C09143=1199.165,141.254,-53.045,-178.295,6.103,148.591
C09144=1199.160,141.502,-53.066,-178.292,6.105,148.590
C09145=1199.155,141.752,-53.087,-178.290,6.105,148.590
C09146=1199.151,142.001,-53.107,-178.287,6.107,148.589
C09147=1199.145,142.250,-53.128,-178.285,6.109,148.589
C09148=1199.141,142.499,-53.148,-178.282,6.110,148.589
C09149=1199.136,142.748,-53.169,-178.279,6.111,148.588
C09150=1199.131,142.997,-53.190,-178.277,6.113,148.588
C09151=1199.127,143.246,-53.210,-178.274,6.114,148.587
C09152=1199.122,143.495,-53.231,-178.272,6.116,148.587
C09153=1199.117,143.744,-53.251,-178.269,6.117,148.586
C09154=1199.112,143.994,-53.272,-178.266,6.118,148.586
C09155=1199.108,144.243,-53.293,-178.264,6.120,148.586
C09156=1199.103,144.492,-53.314,-178.261,6.122,148.585
C09157=1199.099,144.741,-53.335,-178.259,6.122,148.585
C09158=1199.094,144.990,-53.356,-178.256,6.124,148.584
C09159=1199.089,145.239,-53.376,-178.253,6.126,148.584
C09160=1199.084,145.488,-53.397,-178.251,6.126,148.583
C09161=1199.080,145.737,-53.418,-178.248,6.128,148.583
C09162=1199.075,145.986,-53.439,-178.245,6.130,148.582
C09163=1199.070,146.235,-53.459,-178.243,6.132,148.582
C09164=1199.065,146.484,-53.481,-178.240,6.132,148.581
C09165=1199.060,146.733,-53.502,-178.237,6.134,148.581
C09166=1199.056,146.983,-53.522,-178.235,6.136,148.581
C09167=1199.051,147.232,-53.543,-178.232,6.137,148.580
C09168=1199.047,147.481,-53.564,-178.230,6.139,148.580
C09169=1199.042,147.730,-53.585,-178.227,6.140,148.579
C09170=1199.037,147.979,-53.606,-178.224,6.141,148.579
C09171=1199.032,148.228,-53.627,-178.222,6.143,148.578
C09172=1199.027,148.477,-53.648,-178.219,6.145,148.578
C09173=1199.023,148.726,-53.669,-178.217,6.145,148.577
C09174=1199.018,148.976,-53.690,-178.214,6.147,148.577
C09175=1199.013,149.225,-53.711,-178.211,6.149,148.577
C09176=1199.009,149.473,-53.732,-178.208,6.151,148.576
C09177=1199.004,149.722,-53.753,-178.206,6.151,148.576
C09178=1198.999,149.972,-53.774,-178.203,6.153,148.575
C09179=1198.994,150.220,-53.795,-178.201,6.155,148.575
C09180=1198.990,150.470,-53.817,-178.198,6.156,148.575
C09181=1198.985,150.719,-53.838,-178.195,6.157,148.574
C09182=1198.981,150.968,-53.859,-178.193,6.159,148.574
C09183=1198.975,151.217,-53.880,-178.190,6.161,148.573
C09184=1198.970,151.466,-53.901,-178.188,6.162,148.573
C09185=1198.967,151.715,-53.922,-178.185,6.163,148.572
C09186=1198.961,151.964,-53.943,-178.182,6.165,148.572
C09187=1198.957,152.213,-53.965,-178.180,6.166,148.571
C09188=1198.952,152.462,-53.985,-178.177,6.168,148.571
C09189=1198.947,152.711,-54.006,-178.174,6.169,148.571
C09190=1198.943,152.961,-54.028,-178.172,6.171,148.570
C09191=1198.938,153.210,-54.049,-178.169,6.172,148.570
C09192=1198.933,153.458,-54.070,-178.167,6.174,148.569
C09193=1198.928,153.707,-54.091,-178.164,6.175,148.569
C09194=1198.924,153.957,-54.113,-178.161,6.177,148.569
C09195=1198.919,154.206,-54.134,-178.159,6.178,148.568
C09196=1198.914,154.455,-54.156,-178.156,6.180,148.568
C09197=1198.910,154.704,-54.176,-178.153,6.181,148.567
C09198=1198.905,154.953,-54.198,-178.151,6.183,148.567
C09199=1198.900,155.202,-54.219,-178.148,6.184,148.566
C09200=1198.895,155.451,-54.241,-178.146,6.186,148.566
C09201=1198.890,155.699,-54.263,-178.143,6.187,148.565
C09202=1198.887,155.949,-54.283,-178.140,6.189,148.565
C09203=1198.882,156.198,-54.305,-178.138,6.190,148.565
C09204=1198.876,156.447,-54.326,-178.135,6.192,148.564
C09205=1198.872,156.696,-54.348,-178.132,6.194,148.564
C09206=1198.867,156.945,-54.370,-178.129,6.195,148.563
C09207=1198.862,157.194,-54.391,-178.127,6.196,148.563
C09208=1198.858,157.443,-54.412,-178.125,6.198,148.563
C09209=1198.853,157.693,-54.433,-178.122,6.200,148.562
C09210=1198.849,157.941,-54.455,-178.119,6.201,148.562
C09211=1198.844,158.190,-54.476,-178.117,6.202,148.561
C09212=1198.839,158.440,-54.498,-178.114,6.204,148.561
C09213=1198.835,158.708,-54.521,-178.111,6.206,148.560
C09214=1198.829,158.978,-54.545,-178.109,6.207,148.560
C09215=1198.823,159.246,-54.568,-178.105,6.209,148.559
C09216=1198.819,159.515,-54.591,-178.103,6.211,148.559
C09217=1198.814,159.765,-54.612,-178.100,6.212,148.559
C09218=1198.809,160.013,-54.634,-178.097,6.214,148.558
C09219=1198.804,160.262,-54.656,-178.095,6.215,148.558
C09220=1198.800,160.511,-54.678,-178.092,6.217,148.557
C09221=1198.795,160.760,-54.699,-178.089,6.218,148.557
C09222=1198.791,161.010,-54.721,-178.087,6.220,148.557
C09223=1198.786,161.258,-54.743,-178.084,6.222,148.556
C09224=1198.781,161.507,-54.764,-178.082,6.223,148.556
C09225=1198.777,161.756,-54.786,-178.079,6.225,148.556
C09226=1198.771,162.006,-54.807,-178.076,6.226,148.555
C09227=1198.767,162.254,-54.829,-178.073,6.228,148.555
C09228=1198.762,162.504,-54.851,-178.071,6.230,148.554
C09229=1198.757,162.752,-54.873,-178.069,6.231,148.554
C09230=1198.753,163.002,-54.895,-178.066,6.233,148.553
C09231=1198.748,163.250,-54.916,-178.063,6.234,148.553
C09232=1198.744,163.500,-54.938,-178.061,6.236,148.553
C09233=1198.739,163.748,-54.960,-178.058,6.238,148.552
C09234=1198.734,163.998,-54.981,-178.055,6.239,148.552
C09235=1198.730,164.247,-55.003,-178.053,6.240,148.551
C09236=1198.725,164.496,-55.025,-178.050,6.242,148.551
C09237=1198.721,164.745,-55.047,-178.047,6.244,148.551
C09238=1198.716,164.994,-55.069,-178.045,6.246,148.550
C09239=1198.711,165.243,-55.091,-178.043,6.247,148.550
C09240=1198.707,165.492,-55.112,-178.039,6.248,148.549
C09241=1198.702,165.740,-55.134,-178.037,6.250,148.549
C09242=1198.697,165.989,-55.156,-178.034,6.252,148.549
C09243=1198.692,166.238,-55.178,-178.031,6.254,148.548
C09244=1198.688,166.488,-55.200,-178.029,6.255,148.548
C09245=1198.683,166.736,-55.222,-178.027,6.256,148.547
C09246=1198.678,166.986,-55.244,-178.024,6.258,148.547
C09247=1198.674,167.234,-55.266,-178.021,6.260,148.547
C09248=1198.669,167.484,-55.288,-178.019,6.262,148.546
C09249=1198.664,167.732,-55.309,-178.016,6.263,148.546
C09250=1198.660,167.981,-55.333,-178.013,6.264,148.545
C09251=1198.655,168.230,-55.355,-178.011,6.266,148.545
C09252=1198.651,168.479,-55.377,-178.008,6.268,148.545
C09253=1198.646,168.728,-55.398,-178.005,6.270,148.544
C09254=1198.641,168.977,-55.420,-178.003,6.271,148.544
C09255=1198.636,169.226,-55.443,-178.000,6.273,148.544
C09256=1198.632,169.476,-55.465,-177.998,6.274,148.543
C09257=1198.627,169.724,-55.486,-177.995,6.276,148.543
C09258=1198.623,169.973,-55.509,-177.992,6.277,148.542
C09259=1198.618,170.222,-55.531,-177.989,6.279,148.542
C09260=1198.613,170.471,-55.553,-177.987,6.281,148.541
C09261=1198.608,170.720,-55.575,-177.984,6.283,148.541
C09262=1198.604,170.969,-55.597,-177.981,6.285,148.541
C09263=1198.599,171.217,-55.620,-177.979,6.285,148.540
C09264=1198.594,171.467,-55.642,-177.977,6.287,148.540
C09265=1198.590,171.716,-55.664,-177.974,6.289,148.540
C09266=1198.585,171.965,-55.686,-177.971,6.291,148.539
C09267=1198.580,172.214,-55.709,-177.969,6.293,148.539
C09268=1198.575,172.463,-55.731,-177.966,6.294,148.539
C09269=1198.571,172.712,-55.753,-177.963,6.296,148.538
C09270=1198.566,172.961,-55.775,-177.961,6.297,148.538
C09271=1198.562,173.210,-55.798,-177.958,6.299,148.537
C09272=1198.557,173.459,-55.820,-177.955,6.300,148.537
C09273=1198.553,173.708,-55.842,-177.953,6.302,148.536
C09274=1198.548,173.957,-55.865,-177.950,6.304,148.536
C09275=1198.543,174.205,-55.887,-177.947,6.306,148.536
C09276=1198.539,174.455,-55.909,-177.945,6.308,148.535
C09277=1198.534,174.704,-55.932,-177.943,6.309,148.535
C09278=1198.529,174.952,-55.954,-177.940,6.310,148.535
C09279=1198.524,175.201,-55.977,-177.937,6.312,148.534
C09280=1198.520,175.451,-55.999,-177.935,6.314,148.534
C09281=1198.515,175.699,-56.021,-177.932,6.316,148.534
C09282=1198.511,175.948,-56.044,-177.929,6.318,148.533
C09283=1198.506,176.197,-56.066,-177.927,6.319,148.533
C09284=1198.501,176.446,-56.089,-177.924,6.321,148.532
C09285=1198.497,176.695,-56.111,-177.921,6.323,148.532
C09286=1198.492,176.943,-56.134,-177.919,6.324,148.531
C09287=1198.487,177.193,-56.156,-177.916,6.325,148.531
C09288=1198.483,177.442,-56.179,-177.913,6.327,148.531
C09289=1198.478,177.691,-56.201,-177.911,6.329,148.530
C09290=1198.474,177.939,-56.224,-177.908,6.331,148.530
C09291=1198.469,178.189,-56.247,-177.905,6.333,148.530
C09292=1198.464,178.437,-56.269,-177.903,6.334,148.529
C09293=1198.459,178.687,-56.292,-177.900,6.336,148.529
C09294=1198.455,178.935,-56.315,-177.897,6.338,148.529
C09295=1198.450,179.185,-56.337,-177.895,6.340,148.528
C09296=1198.446,179.433,-56.360,-177.893,6.341,148.528
C09297=1198.441,179.682,-56.382,-177.890,6.343,148.528
C09298=1198.437,179.932,-56.405,-177.887,6.344,148.527
C09299=1198.431,180.180,-56.428,-177.885,6.346,148.527
C09300=1198.427,180.429,-56.450,-177.882,6.348,148.526
C09301=1198.422,180.678,-56.474,-177.879,6.350,148.526
C09302=1198.418,180.927,-56.496,-177.877,6.352,148.526
C09303=1198.413,181.176,-56.519,-177.874,6.353,148.525
C09304=1198.409,181.425,-56.541,-177.871,6.355,148.525
C09305=1198.404,181.674,-56.565,-177.869,6.357,148.525
C09306=1198.400,181.923,-56.587,-177.866,6.359,148.524
C09307=1198.394,182.171,-56.610,-177.863,6.361,148.524
C09308=1198.391,182.420,-56.633,-177.861,6.362,148.524
C09309=1198.386,182.670,-56.655,-177.859,6.363,148.523
C09310=1198.381,182.919,-56.679,-177.856,6.365,148.523
C09311=1198.376,183.167,-56.701,-177.853,6.367,148.522
C09312=1198.372,183.416,-56.724,-177.851,6.369,148.522
C09313=1198.367,183.665,-56.746,-177.848,6.371,148.522
C09314=1198.363,183.914,-56.770,-177.845,6.373,148.521
C09315=1198.358,184.163,-56.793,-177.843,6.374,148.521
C09316=1198.353,184.411,-56.815,-177.840,6.376,148.521
C09317=1198.348,184.681,-56.840,-177.837,6.378,148.520
C09318=1198.343,184.951,-56.866,-177.834,6.379,148.520
C09319=1198.338,185.220,-56.890,-177.831,6.381,148.519
C09320=1198.333,185.490,-56.915,-177.828,6.384,148.519
C09321=1198.328,185.739,-56.938,-177.826,6.386,148.519
C09322=1198.324,185.988,-56.961,-177.823,6.387,148.518
C09323=1198.319,186.237,-56.984,-177.820,6.389,148.518
C09324=1198.315,186.486,-57.008,-177.818,6.390,148.518
C09325=1198.310,186.734,-57.030,-177.816,6.392,148.517
C09326=1198.305,186.983,-57.053,-177.813,6.394,148.517
C09327=1198.300,187.232,-57.076,-177.810,6.396,148.517
C09328=1198.296,187.482,-57.100,-177.808,6.397,148.516
C09329=1198.292,187.730,-57.122,-177.805,6.399,148.516
C09330=1198.287,187.979,-57.146,-177.802,6.401,148.516
C09331=1198.282,188.228,-57.169,-177.800,6.403,148.515
C09332=1198.277,188.477,-57.192,-177.797,6.405,148.515
C09333=1198.273,188.725,-57.215,-177.794,6.406,148.514
C09334=1198.268,188.974,-57.238,-177.792,6.408,148.514
C09335=1198.264,189.223,-57.262,-177.789,6.410,148.514
C09336=1198.259,189.472,-57.285,-177.786,6.412,148.513
C09337=1198.255,189.721,-57.308,-177.784,6.414,148.513
C09338=1198.250,189.970,-57.331,-177.781,6.416,148.513
C09339=1198.246,190.219,-57.354,-177.778,6.417,148.512
C09340=1198.241,190.468,-57.378,-177.776,6.419,148.512
C09341=1198.236,190.717,-57.401,-177.773,6.421,148.512
C09342=1198.231,190.966,-57.424,-177.771,6.423,148.512
C09343=1198.227,191.214,-57.447,-177.768,6.425,148.511
C09344=1198.222,191.463,-57.470,-177.765,6.427,148.511
C09345=1198.218,191.712,-57.494,-177.763,6.429,148.511
C09346=1198.213,191.961,-57.518,-177.760,6.430,148.510
C09347=1198.209,192.210,-57.541,-177.757,6.432,148.510
C09348=1198.204,192.459,-57.564,-177.755,6.434,148.509
C09349=1198.199,192.708,-57.588,-177.752,6.436,148.509
C09350=1198.194,192.957,-57.611,-177.750,6.438,148.509
C09351=1198.190,193.206,-57.634,-177.747,6.439,148.508
C09352=1198.186,193.454,-57.658,-177.744,6.441,148.508
C09353=1198.181,193.703,-57.681,-177.742,6.443,148.508
C09354=1198.177,193.952,-57.705,-177.739,6.445,148.507
C09355=1198.172,194.201,-57.728,-177.736,6.447,148.507
C09356=1198.168,194.450,-57.752,-177.734,6.448,148.507
C09357=1198.163,194.699,-57.775,-177.731,6.450,148.506
C09358=1198.158,194.948,-57.799,-177.728,6.452,148.506
C09359=1198.153,195.197,-57.822,-177.726,6.454,148.506
C09360=1198.149,195.445,-57.846,-177.723,6.456,148.505
C09361=1198.144,195.694,-57.870,-177.721,6.458,148.505
C09362=1198.140,195.943,-57.893,-177.718,6.460,148.505
C09363=1198.135,196.192,-57.917,-177.715,6.461,148.504
C09364=1198.131,196.441,-57.940,-177.713,6.463,148.504
C09365=1198.126,196.690,-57.964,-177.710,6.465,148.504
C09366=1198.121,196.938,-57.988,-177.707,6.467,148.503
C09367=1198.117,197.187,-58.011,-177.705,6.469,148.503
C09368=1198.112,197.436,-58.035,-177.702,6.471,148.503
C09369=1198.108,197.685,-58.059,-177.700,6.472,148.502
C09370=1198.103,197.934,-58.082,-177.697,6.474,148.502
C09371=1198.098,198.183,-58.105,-177.695,6.476,148.502
C09372=1198.094,198.431,-58.129,-177.692,6.478,148.502
C09373=1198.089,198.680,-58.153,-177.689,6.480,148.501
C09374=1198.085,198.928,-58.177,-177.687,6.482,148.501
C09375=1198.080,199.177,-58.200,-177.684,6.484,148.501
C09376=1198.076,199.426,-58.224,-177.681,6.485,148.500
C09377=1198.070,199.675,-58.248,-177.679,6.487,148.500
C09378=1198.066,199.924,-58.272,-177.676,6.490,148.500
C09379=1198.061,200.173,-58.296,-177.673,6.492,148.499
C09380=1198.057,200.421,-58.320,-177.670,6.493,148.499
C09381=1198.053,200.671,-58.343,-177.668,6.496,148.499
C09382=1198.048,200.919,-58.368,-177.665,6.497,148.498
C09383=1198.044,201.168,-58.391,-177.663,6.499,148.498
C09384=1198.039,201.417,-58.415,-177.660,6.501,148.498
C09385=1198.034,201.666,-58.439,-177.657,6.503,148.497
C09386=1198.029,201.914,-58.463,-177.655,6.505,148.497
C09387=1198.025,202.163,-58.486,-177.652,6.506,148.497
C09388=1198.020,202.412,-58.510,-177.649,6.508,148.496
C09389=1198.016,202.661,-58.535,-177.647,6.510,148.496
C09390=1198.012,202.910,-58.558,-177.645,6.512,148.496
C09391=1198.007,203.159,-58.583,-177.642,6.514,148.495
C09392=1198.002,203.408,-58.606,-177.639,6.516,148.495
C09393=1197.998,203.656,-58.630,-177.637,6.518,148.495
C09394=1197.993,203.905,-58.654,-177.634,6.520,148.494
C09395=1197.988,204.154,-58.678,-177.631,6.522,148.494
C09396=1197.984,204.403,-58.703,-177.628,6.524,148.494
C09397=1197.980,204.652,-58.727,-177.626,6.526,148.494
C09398=1197.975,204.900,-58.751,-177.623,6.528,148.493
C09399=1197.970,205.149,-58.775,-177.621,6.530,148.493
C09400=1197.965,205.398,-58.799,-177.618,6.532,148.493
C09401=1197.962,205.647,-58.823,-177.615,6.533,148.492
C09402=1197.957,205.896,-58.847,-177.613,6.535,148.492
C09403=1197.952,206.145,-58.871,-177.610,6.537,148.492
C09404=1197.947,206.393,-58.896,-177.608,6.539,148.492
C09405=1197.943,206.641,-58.920,-177.605,6.541,148.491
C09406=1197.938,206.891,-58.945,-177.602,6.544,148.491
C09407=1197.934,207.140,-58.968,-177.599,6.545,148.491
C09408=1197.929,207.388,-58.992,-177.597,6.547,148.490
C09409=1197.924,207.637,-59.017,-177.594,6.549,148.490
C09410=1197.920,207.885,-59.041,-177.592,6.551,148.490
C09411=1197.916,208.134,-59.065,-177.589,6.553,148.489
C09412=1197.911,208.383,-59.090,-177.587,6.555,148.489
C09413=1197.906,208.632,-59.113,-177.584,6.557,148.489
C09414=1197.902,208.881,-59.137,-177.581,6.559,148.488
C09415=1197.897,209.130,-59.162,-177.579,6.560,148.488
C09416=1197.893,209.378,-59.186,-177.576,6.563,148.488
C09417=1197.888,209.627,-59.211,-177.573,6.565,148.488
C09418=1197.883,209.876,-59.235,-177.571,6.567,148.487
C09419=1197.879,210.125,-59.260,-177.568,6.569,148.487
C09420=1197.874,210.373,-59.284,-177.565,6.571,148.487
C09421=1197.869,210.644,-59.311,-177.563,6.572,148.486
C09422=1197.864,210.914,-59.336,-177.559,6.575,148.486
C09423=1197.860,211.185,-59.363,-177.557,6.577,148.486
C09424=1197.855,211.455,-59.390,-177.554,6.580,148.485
C09425=1197.850,211.704,-59.415,-177.551,6.582,148.485
C09426=1197.845,211.952,-59.439,-177.549,6.584,148.485
C09427=1197.841,212.202,-59.464,-177.546,6.585,148.485
C09428=1197.836,212.450,-59.488,-177.544,6.587,148.484
C09429=1197.831,212.699,-59.513,-177.541,6.589,148.484
C09430=1197.827,212.948,-59.537,-177.539,6.591,148.484
C09431=1197.822,213.197,-59.562,-177.536,6.593,148.483
C09432=1197.818,213.445,-59.586,-177.533,6.596,148.483
C09433=1197.814,213.694,-59.612,-177.530,6.597,148.483
C09434=1197.809,213.942,-59.636,-177.528,6.599,148.482
C09435=1197.804,214.191,-59.660,-177.525,6.601,148.482
C09436=1197.800,214.440,-59.685,-177.523,6.603,148.482
C09437=1197.795,214.689,-59.710,-177.520,6.605,148.482
C09438=1197.791,214.938,-59.734,-177.517,6.607,148.481
C09439=1197.786,215.187,-59.759,-177.514,6.610,148.481
C09440=1197.782,215.434,-59.783,-177.512,6.612,148.481
C09441=1197.778,215.684,-59.808,-177.509,6.614,148.481
C09442=1197.773,215.933,-59.833,-177.507,6.615,148.480
C09443=1197.768,216.181,-59.857,-177.504,6.617,148.480
C09444=1197.764,216.430,-59.882,-177.501,6.619,148.480
C09445=1197.760,216.678,-59.907,-177.499,6.622,148.479
C09446=1197.755,216.928,-59.932,-177.496,6.624,148.479
C09447=1197.750,217.176,-59.957,-177.493,6.626,148.479
C09448=1197.746,217.424,-59.982,-177.491,6.627,148.478
C09449=1197.741,217.674,-60.007,-177.489,6.630,148.478
C09450=1197.736,217.922,-60.031,-177.486,6.631,148.478
C09451=1197.732,218.171,-60.056,-177.483,6.634,148.478
C09452=1197.727,218.420,-60.081,-177.480,6.636,148.477
C09453=1197.723,218.669,-60.106,-177.478,6.638,148.477
C09454=1197.719,218.917,-60.130,-177.475,6.640,148.477
C09455=1197.714,219.166,-60.156,-177.473,6.642,148.477
C09456=1197.709,219.415,-60.181,-177.470,6.644,148.476
C09457=1197.705,219.663,-60.205,-177.467,6.647,148.476
C09458=1197.701,219.912,-60.230,-177.465,6.648,148.476
C09459=1197.695,220.161,-60.255,-177.462,6.650,148.476
C09460=1197.692,220.409,-60.280,-177.459,6.652,148.475
C09461=1197.687,220.658,-60.305,-177.457,6.654,148.475
C09462=1197.683,220.907,-60.331,-177.455,6.656,148.475
C09463=1197.677,221.156,-60.355,-177.451,6.659,148.474
C09464=1197.674,221.404,-60.380,-177.449,6.660,148.474
C09465=1197.669,221.653,-60.405,-177.447,6.663,148.474
C09466=1197.664,221.902,-60.430,-177.444,6.664,148.474
C09467=1197.660,222.150,-60.456,-177.441,6.666,148.473
C09468=1197.655,222.400,-60.481,-177.438,6.669,148.473
C09469=1197.651,222.648,-60.505,-177.436,6.671,148.473
C09470=1197.647,222.896,-60.531,-177.433,6.673,148.473
C09471=1197.642,223.145,-60.556,-177.431,6.675,148.472
C09472=1197.637,223.394,-60.582,-177.428,6.677,148.472
C09473=1197.632,223.643,-60.606,-177.426,6.679,148.472
C09474=1197.629,223.891,-60.631,-177.423,6.681,148.472
C09475=1197.624,224.140,-60.656,-177.420,6.683,148.471
C09476=1197.619,224.389,-60.682,-177.418,6.685,148.471
C09477=1197.615,224.637,-60.707,-177.415,6.687,148.471
C09478=1197.610,224.886,-60.732,-177.412,6.689,148.470
C09479=1197.606,225.135,-60.758,-177.410,6.692,148.470
C09480=1197.601,225.384,-60.783,-177.407,6.694,148.470
C09481=1197.597,225.632,-60.808,-177.404,6.696,148.470
C09482=1197.592,225.880,-60.833,-177.402,6.698,148.470
C09483=1197.588,226.130,-60.858,-177.400,6.700,148.469
C09484=1197.583,226.378,-60.884,-177.396,6.702,148.469
C09485=1197.579,226.627,-60.909,-177.394,6.704,148.469
C09486=1197.574,226.875,-60.935,-177.392,6.706,148.469
C09487=1197.569,227.124,-60.960,-177.389,6.708,148.468
C09488=1197.565,227.373,-60.986,-177.386,6.711,148.468
C09489=1197.560,227.621,-61.011,-177.384,6.713,148.468
C09490=1197.556,227.871,-61.036,-177.381,6.715,148.468
C09491=1197.552,228.119,-61.062,-177.378,6.717,148.467
C09492=1197.547,228.367,-61.087,-177.376,6.719,148.467
C09493=1197.543,228.616,-61.113,-177.373,6.721,148.467
C09494=1197.538,228.864,-61.138,-177.370,6.723,148.466
C09495=1197.533,229.114,-61.163,-177.368,6.725,148.466
C09496=1197.529,229.363,-61.189,-177.366,6.727,148.466
C09497=1197.524,229.611,-61.214,-177.363,6.729,148.466
C09498=1197.520,229.859,-61.240,-177.360,6.732,148.466
C09499=1197.516,230.108,-61.266,-177.358,6.734,148.465
C09500=1197.511,230.356,-61.291,-177.355,6.736,148.465
C09501=1197.507,230.605,-61.317,-177.353,6.738,148.465
C09502=1197.502,230.854,-61.343,-177.350,6.741,148.465
C09503=1197.497,231.103,-61.367,-177.347,6.742,148.464
C09504=1197.493,231.352,-61.393,-177.345,6.745,148.464
C09505=1197.489,231.600,-61.419,-177.342,6.746,148.464
C09506=1197.484,231.848,-61.444,-177.339,6.749,148.464
C09507=1197.480,232.097,-61.470,-177.337,6.751,148.463
C09508=1197.476,232.346,-61.496,-177.334,6.753,148.463
C09509=1197.471,232.594,-61.521,-177.332,6.755,148.463
C09510=1197.466,232.843,-61.547,-177.329,6.758,148.463
C09511=1197.461,233.092,-61.573,-177.326,6.760,148.462
C09512=1197.457,233.341,-61.599,-177.324,6.762,148.462
C09513=1197.452,233.589,-61.624,-177.321,6.764,148.462
C09514=1197.448,233.838,-61.650,-177.319,6.767,148.462
C09515=1197.444,234.087,-61.676,-177.316,6.769,148.462
C09516=1197.439,234.335,-61.701,-177.313,6.770,148.461
C09517=1197.435,234.583,-61.727,-177.311,6.773,148.461
C09518=1197.430,234.833,-61.753,-177.308,6.775,148.461
C09519=1197.426,235.081,-61.780,-177.305,6.777,148.461
C09520=1197.421,235.329,-61.805,-177.303,6.779,148.460
C09521=1197.417,235.578,-61.831,-177.301,6.781,148.460
C09522=1197.413,235.827,-61.857,-177.298,6.784,148.460
C09523=1197.408,236.076,-61.883,-177.295,6.786,148.460
C09524=1197.403,236.324,-61.909,-177.293,6.788,148.459
C09525=1197.399,236.595,-61.937,-177.290,6.791,148.459
C09526=1197.394,236.867,-61.965,-177.287,6.793,148.459
C09527=1197.389,237.139,-61.993,-177.284,6.795,148.459
C09528=1197.384,237.410,-62.022,-177.282,6.797,148.459
C09529=1197.379,237.659,-62.048,-177.279,6.800,148.458
C09530=1197.375,237.907,-62.074,-177.276,6.802,148.458
C09531=1197.371,238.155,-62.100,-177.274,6.804,148.458
C09532=1197.366,238.404,-62.126,-177.271,6.807,148.458
C09533=1197.361,238.653,-62.152,-177.268,6.809,148.458
C09534=1197.357,238.902,-62.178,-177.266,6.811,148.457
C09535=1197.352,239.150,-62.205,-177.263,6.812,148.457
C09536=1197.348,239.399,-62.231,-177.260,6.815,148.457
C09537=1197.344,239.648,-62.256,-177.258,6.817,148.457
C09538=1197.340,239.895,-62.282,-177.256,6.819,148.456
C09539=1197.335,240.144,-62.309,-177.252,6.822,148.456
C09540=1197.330,240.393,-62.335,-177.250,6.824,148.456
C09541=1197.326,240.642,-62.362,-177.248,6.826,148.456
C09542=1197.321,240.890,-62.387,-177.245,6.828,148.456
C09543=1197.317,241.139,-62.413,-177.242,6.831,148.455
C09544=1197.313,241.388,-62.440,-177.240,6.833,148.455
C09545=1197.308,241.636,-62.466,-177.238,6.835,148.455
C09546=1197.304,241.884,-62.492,-177.234,6.838,148.455
C09547=1197.299,242.133,-62.518,-177.232,6.840,148.455
C09548=1197.295,242.382,-62.544,-177.230,6.842,148.454
C09549=1197.290,242.630,-62.571,-177.227,6.845,148.454
C09550=1197.286,242.879,-62.597,-177.224,6.846,148.454
C09551=1197.282,243.127,-62.623,-177.222,6.849,148.454
C09552=1197.277,243.376,-62.650,-177.219,6.851,148.454
C09553=1197.273,243.625,-62.676,-177.217,6.853,148.453
C09554=1197.267,243.873,-62.702,-177.214,6.855,148.453
C09555=1197.263,244.121,-62.729,-177.212,6.857,148.453
C09556=1197.258,244.370,-62.755,-177.209,6.860,148.453
C09557=1197.255,244.619,-62.781,-177.207,6.862,148.453
C09558=1197.250,244.868,-62.808,-177.204,6.864,148.452
C09559=1197.246,245.116,-62.834,-177.201,6.867,148.452
C09560=1197.241,245.364,-62.861,-177.199,6.869,148.452
C09561=1197.237,245.613,-62.887,-177.196,6.871,148.452
C09562=1197.232,245.862,-62.914,-177.193,6.874,148.452
C09563=1197.228,246.110,-62.940,-177.191,6.876,148.451
C09564=1197.223,246.359,-62.967,-177.188,6.878,148.451
C09565=1197.219,246.607,-62.993,-177.185,6.881,148.451
C09566=1197.214,246.856,-63.020,-177.183,6.883,148.451
C09567=1197.210,247.104,-63.046,-177.180,6.885,148.450
C09568=1197.206,247.353,-63.073,-177.178,6.888,148.450
C09569=1197.202,247.602,-63.099,-177.175,6.889,148.450
C09570=1197.197,247.850,-63.126,-177.173,6.892,148.450
C09571=1197.192,248.099,-63.153,-177.170,6.894,148.450
C09572=1197.188,248.348,-63.179,-177.168,6.896,148.450
C09573=1197.183,248.596,-63.206,-177.164,6.899,148.449
C09574=1197.179,248.844,-63.232,-177.162,6.901,148.449
C09575=1197.175,249.093,-63.260,-177.160,6.903,148.449
C09576=1197.170,249.342,-63.286,-177.157,6.906,148.449
C09577=1197.166,249.590,-63.312,-177.155,6.908,148.449
C09578=1197.161,249.838,-63.339,-177.152,6.910,148.449
C09579=1197.157,250.087,-63.366,-177.149,6.913,148.448
C09580=1197.153,250.335,-63.393,-177.147,6.915,148.448
C09581=1197.148,250.584,-63.420,-177.145,6.917,148.448
C09582=1197.143,250.833,-63.446,-177.141,6.920,148.448
C09583=1197.139,251.081,-63.473,-177.139,6.922,148.448
C09584=1197.135,251.329,-63.500,-177.137,6.924,148.447
C09585=1197.130,251.578,-63.527,-177.134,6.927,148.447
C09586=1197.126,251.826,-63.553,-177.131,6.929,148.447
C09587=1197.121,252.075,-63.580,-177.129,6.932,148.447
C09588=1197.117,252.323,-63.608,-177.126,6.934,148.447
C09589=1197.112,252.572,-63.635,-177.124,6.936,148.447
C09590=1197.109,252.820,-63.661,-177.121,6.939,148.446
C09591=1197.104,253.070,-63.688,-177.118,6.940,148.446
C09592=1197.099,253.318,-63.715,-177.116,6.943,148.446
C09593=1197.095,253.566,-63.741,-177.113,6.945,148.446
C09594=1197.090,253.815,-63.768,-177.111,6.947,148.446
C09595=1197.086,254.063,-63.795,-177.108,6.950,148.445
C09596=1197.081,254.312,-63.822,-177.106,6.952,148.445
C09597=1197.076,254.560,-63.850,-177.103,6.954,148.445
C09598=1197.073,254.808,-63.876,-177.100,6.957,148.445
C09599=1197.069,255.058,-63.903,-177.098,6.959,148.445
C09600=1197.064,255.306,-63.931,-177.095,6.962,148.445
C09601=1197.060,255.554,-63.958,-177.093,6.964,148.445
C09602=1197.055,255.803,-63.985,-177.090,6.966,148.444
C09603=1197.051,256.051,-64.012,-177.087,6.969,148.444
C09604=1197.046,256.299,-64.039,-177.085,6.971,148.444
C09605=1197.042,256.548,-64.066,-177.082,6.974,148.444
C09606=1197.038,256.797,-64.093,-177.080,6.976,148.444
C09607=1197.033,257.045,-64.120,-177.077,6.978,148.443
C09608=1197.028,257.294,-64.147,-177.075,6.981,148.443
C09609=1197.024,257.542,-64.175,-177.072,6.983,148.443
C09610=1197.019,257.790,-64.202,-177.069,6.986,148.443
C09611=1197.015,258.038,-64.229,-177.067,6.988,148.443
C09612=1197.011,258.288,-64.256,-177.064,6.991,148.443
C09613=1197.007,258.536,-64.283,-177.062,6.993,148.443
C09614=1197.002,258.784,-64.311,-177.060,6.995,148.443
C09615=1196.998,259.032,-64.338,-177.056,6.998,148.442
C09616=1196.993,259.281,-64.365,-177.054,7.000,148.442
C09617=1196.989,259.530,-64.393,-177.051,7.003,148.442
C09618=1196.985,259.778,-64.420,-177.049,7.005,148.442
C09619=1196.980,260.027,-64.447,-177.046,7.008,148.442
C09620=1196.975,260.275,-64.474,-177.044,7.009,148.441
C09621=1196.971,260.524,-64.502,-177.041,7.012,148.441
C09622=1196.967,260.772,-64.530,-177.039,7.015,148.441
C09623=1196.962,261.021,-64.557,-177.036,7.016,148.441
C09624=1196.958,261.269,-64.584,-177.033,7.019,148.441
C09625=1196.954,261.518,-64.612,-177.031,7.022,148.441
C09626=1196.949,261.766,-64.639,-177.028,7.024,148.441
C09627=1196.945,262.014,-64.667,-177.026,7.026,148.441
C09628=1196.940,262.263,-64.694,-177.023,7.029,148.440
C09629=1196.935,262.536,-64.725,-177.020,7.031,148.440
C09630=1196.931,262.808,-64.754,-177.017,7.034,148.440
C09631=1196.926,263.081,-64.785,-177.015,7.037,148.440
C09632=1196.921,263.354,-64.815,-177.012,7.040,148.440
C09633=1196.916,263.603,-64.842,-177.009,7.042,148.440
C09634=1196.912,263.851,-64.870,-177.007,7.045,148.439
C09635=1196.908,264.100,-64.898,-177.004,7.047,148.439
C09636=1196.904,264.348,-64.925,-177.001,7.050,148.439
C09637=1196.899,264.596,-64.952,-176.999,7.052,148.439
C09638=1196.895,264.845,-64.980,-176.997,7.054,148.439
C09639=1196.890,265.093,-65.008,-176.994,7.057,148.439
C09640=1196.886,265.341,-65.035,-176.992,7.059,148.439
C09641=1196.881,265.591,-65.063,-176.989,7.062,148.439
C09642=1196.877,265.838,-65.091,-176.986,7.064,148.438
C09643=1196.872,266.087,-65.118,-176.984,7.067,148.438
C09644=1196.869,266.335,-65.146,-176.981,7.069,148.438
C09645=1196.864,266.583,-65.174,-176.978,7.072,148.438
C09646=1196.860,266.832,-65.201,-176.976,7.074,148.438
C09647=1196.855,267.081,-65.230,-176.973,7.077,148.438
C09648=1196.850,267.329,-65.257,-176.971,7.079,148.437
C09649=1196.846,267.577,-65.285,-176.968,7.082,148.437
C09650=1196.842,267.826,-65.313,-176.966,7.084,148.437
C09651=1196.838,268.074,-65.340,-176.963,7.086,148.437
C09652=1196.833,268.323,-65.369,-176.961,7.089,148.437
C09653=1196.829,268.571,-65.396,-176.958,7.092,148.437
C09654=1196.824,268.819,-65.424,-176.956,7.094,148.437
C09655=1196.820,269.068,-65.452,-176.952,7.097,148.437
C09656=1196.815,269.316,-65.480,-176.950,7.099,148.437
C09657=1196.811,269.564,-65.508,-176.948,7.102,148.436
C09658=1196.807,269.813,-65.536,-176.945,7.104,148.436
C09659=1196.803,270.061,-65.563,-176.942,7.107,148.436
C09660=1196.798,270.310,-65.592,-176.940,7.109,148.436
C09661=1196.794,270.558,-65.620,-176.937,7.112,148.436
C09662=1196.790,270.807,-65.648,-176.935,7.114,148.436
C09663=1196.785,271.055,-65.676,-176.932,7.117,148.436
C09664=1196.780,271.303,-65.703,-176.930,7.119,148.436
C09665=1196.777,271.552,-65.731,-176.927,7.121,148.435
C09666=1196.771,271.800,-65.760,-176.925,7.124,148.435
C09667=1196.768,272.049,-65.788,-176.922,7.127,148.435
C09668=1196.763,272.296,-65.816,-176.920,7.129,148.435
C09669=1196.759,272.545,-65.844,-176.917,7.131,148.435
C09670=1196.754,272.793,-65.872,-176.914,7.134,148.435
C09671=1196.751,273.042,-65.900,-176.912,7.137,148.435
C09672=1196.745,273.291,-65.928,-176.910,7.139,148.435
C09673=1196.742,273.539,-65.956,-176.906,7.142,148.434
C09674=1196.737,273.787,-65.984,-176.904,7.144,148.434
C09675=1196.733,274.036,-66.013,-176.902,7.147,148.434
C09676=1196.728,274.284,-66.040,-176.899,7.149,148.434
C09677=1196.724,274.533,-66.069,-176.896,7.152,148.434
C09678=1196.720,274.781,-66.097,-176.894,7.154,148.434
C09679=1196.715,275.029,-66.126,-176.891,7.157,148.434
C09680=1196.711,275.277,-66.153,-176.889,7.160,148.434
C09681=1196.706,275.526,-66.182,-176.886,7.162,148.434
C09682=1196.702,275.774,-66.210,-176.883,7.165,148.434
C09683=1196.698,276.022,-66.239,-176.881,7.167,148.433
C09684=1196.693,276.270,-66.267,-176.878,7.170,148.433
C09685=1196.689,276.519,-66.296,-176.876,7.172,148.433
C09686=1196.685,276.768,-66.324,-176.873,7.175,148.433
C09687=1196.680,277.016,-66.352,-176.871,7.177,148.433
C09688=1196.676,277.264,-66.380,-176.868,7.180,148.433
C09689=1196.671,277.513,-66.409,-176.866,7.182,148.433
C09690=1196.667,277.761,-66.437,-176.863,7.185,148.433
C09691=1196.663,278.009,-66.466,-176.860,7.188,148.433
C09692=1196.659,278.257,-66.494,-176.858,7.190,148.433
C09693=1196.654,278.506,-66.523,-176.855,7.193,148.432
C09694=1196.650,278.754,-66.551,-176.853,7.195,148.432
C09695=1196.646,279.003,-66.579,-176.851,7.198,148.432
C09696=1196.642,279.250,-66.608,-176.848,7.200,148.432
C09697=1196.637,279.499,-66.637,-176.845,7.203,148.432
C09698=1196.633,279.748,-66.665,-176.843,7.205,148.432
C09699=1196.628,279.996,-66.693,-176.840,7.208,148.432
C09700=1196.624,280.244,-66.723,-176.838,7.211,148.432
C09701=1196.620,280.492,-66.750,-176.835,7.213,148.432
C09702=1196.615,280.741,-66.779,-176.832,7.216,148.432
C09703=1196.611,280.989,-66.809,-176.830,7.218,148.431
C09704=1196.607,281.237,-66.836,-176.827,7.221,148.431
C09705=1196.602,281.486,-66.865,-176.825,7.223,148.431
C09706=1196.598,281.734,-66.895,-176.823,7.226,148.431
C09707=1196.594,281.982,-66.922,-176.819,7.229,148.431
C09708=1196.589,282.231,-66.951,-176.817,7.231,148.431
C09709=1196.585,282.479,-66.981,-176.815,7.234,148.431
C09710=1196.581,282.727,-67.008,-176.812,7.236,148.431
C09711=1196.576,282.976,-67.037,-176.810,7.239,148.431
C09712=1196.572,283.224,-67.067,-176.807,7.242,148.431
C09713=1196.568,283.472,-67.094,-176.805,7.245,148.431
C09714=1196.563,283.720,-67.124,-176.802,7.247,148.431
C09715=1196.559,283.969,-67.152,-176.800,7.249,148.430
C09716=1196.554,284.217,-67.182,-176.797,7.253,148.430
C09717=1196.550,284.465,-67.210,-176.794,7.256,148.430
C09718=1196.546,284.714,-67.239,-176.792,7.258,148.430
C09719=1196.541,284.962,-67.268,-176.789,7.261,148.430
C09720=1196.537,285.210,-67.297,-176.787,7.263,148.430
C09721=1196.533,285.459,-67.325,-176.784,7.266,148.430
C09722=1196.529,285.707,-67.355,-176.781,7.269,148.430
C09723=1196.524,285.955,-67.383,-176.779,7.271,148.430
C09724=1196.520,286.203,-67.412,-176.776,7.274,148.430
C09725=1196.516,286.452,-67.442,-176.774,7.276,148.430
C09726=1196.512,286.700,-67.470,-176.772,7.279,148.430
C09727=1196.507,286.948,-67.499,-176.769,7.282,148.430
C09728=1196.503,287.197,-67.528,-176.767,7.284,148.430
C09729=1196.498,287.445,-67.557,-176.764,7.287,148.430
C09730=1196.494,287.693,-67.587,-176.762,7.289,148.430
C09731=1196.489,287.941,-67.615,-176.759,7.292,148.429
C09732=1196.485,288.190,-67.645,-176.756,7.295,148.429
C09733=1196.480,288.464,-67.676,-176.753,7.298,148.429
C09734=1196.476,288.739,-67.709,-176.751,7.301,148.429
C09735=1196.471,289.013,-67.741,-176.748,7.304,148.429
C09736=1196.466,289.288,-67.773,-176.745,7.307,148.429
C09737=1196.462,289.536,-67.802,-176.743,7.309,148.429
C09738=1196.457,289.784,-67.832,-176.740,7.312,148.429
C09739=1196.453,290.032,-67.861,-176.737,7.315,148.429
C09740=1196.449,290.280,-67.889,-176.735,7.317,148.429
C09741=1196.445,290.529,-67.918,-176.732,7.320,148.429
C09742=1196.441,290.777,-67.948,-176.730,7.322,148.429
C09743=1196.436,291.025,-67.977,-176.727,7.325,148.429
C09744=1196.432,291.273,-68.007,-176.725,7.328,148.429
C09745=1196.428,291.522,-68.036,-176.723,7.331,148.429
C09746=1196.423,291.770,-68.065,-176.720,7.334,148.429
C09747=1196.419,292.018,-68.094,-176.717,7.337,148.429
C09748=1196.415,292.266,-68.124,-176.715,7.339,148.428
C09749=1196.410,292.515,-68.153,-176.712,7.342,148.428
C09750=1196.406,292.763,-68.182,-176.710,7.345,148.428
C09751=1196.402,293.011,-68.212,-176.708,7.347,148.428
C09752=1196.398,293.259,-68.241,-176.705,7.350,148.428
C09753=1196.393,293.507,-68.270,-176.703,7.352,148.428
C09754=1196.389,293.755,-68.300,-176.700,7.355,148.428
C09755=1196.385,294.003,-68.329,-176.697,7.358,148.428
C09756=1196.381,294.252,-68.359,-176.695,7.360,148.428
C09757=1196.376,294.500,-68.389,-176.692,7.363,148.428
C09758=1196.371,294.749,-68.418,-176.689,7.366,148.428
C09759=1196.367,294.997,-68.448,-176.687,7.368,148.428
C09760=1196.363,295.245,-68.477,-176.684,7.371,148.428
C09761=1196.359,295.493,-68.507,-176.682,7.374,148.428
C09762=1196.355,295.742,-68.536,-176.680,7.376,148.428
C09763=1196.351,295.990,-68.566,-176.677,7.379,148.428
C09764=1196.346,296.238,-68.595,-176.674,7.382,148.428
C09765=1196.342,296.486,-68.624,-176.672,7.385,148.428
C09766=1196.337,296.734,-68.654,-176.669,7.388,148.428
C09767=1196.332,296.983,-68.684,-176.667,7.391,148.428
C09768=1196.328,297.231,-68.713,-176.665,7.393,148.427
C09769=1196.324,297.479,-68.743,-176.662,7.396,148.427
C09770=1196.320,297.727,-68.773,-176.659,7.399,148.427
C09771=1196.316,297.975,-68.802,-176.657,7.401,148.427
C09772=1196.311,298.224,-68.832,-176.655,7.404,148.428
C09773=1196.307,298.472,-68.862,-176.652,7.407,148.428
C09774=1196.303,298.720,-68.891,-176.650,7.410,148.427
C09775=1196.299,298.968,-68.921,-176.647,7.413,148.427
C09776=1196.295,299.216,-68.951,-176.644,7.416,148.427
C09777=1196.290,299.465,-68.981,-176.642,7.418,148.427
C09778=1196.286,299.713,-69.010,-176.640,7.421,148.427
C09779=1196.282,299.961,-69.040,-176.637,7.424,148.427
C09780=1196.278,300.209,-69.070,-176.635,7.426,148.427
C09781=1196.273,300.457,-69.100,-176.632,7.429,148.427
C09782=1196.269,300.705,-69.130,-176.629,7.432,148.427
C09783=1196.265,300.953,-69.159,-176.627,7.435,148.427
C09784=1196.260,301.202,-69.189,-176.625,7.437,148.427
C09785=1196.256,301.450,-69.220,-176.622,7.440,148.427
C09786=1196.252,301.698,-69.249,-176.619,7.443,148.427
C09787=1196.247,301.946,-69.279,-176.617,7.445,148.427
C09788=1196.243,302.194,-69.309,-176.614,7.448,148.427
C09789=1196.239,302.442,-69.339,-176.612,7.451,148.427
C09790=1196.234,302.691,-69.368,-176.610,7.454,148.427
C09791=1196.230,302.939,-69.399,-176.607,7.457,148.427
C09792=1196.226,303.188,-69.429,-176.605,7.460,148.427
C09793=1196.222,303.435,-69.460,-176.602,7.462,148.427
C09794=1196.217,303.684,-69.489,-176.600,7.465,148.427
C09795=1196.214,303.931,-69.519,-176.597,7.468,148.427
C09796=1196.209,304.180,-69.549,-176.594,7.471,148.427
C09797=1196.205,304.428,-69.579,-176.592,7.473,148.427
C09798=1196.201,304.676,-69.609,-176.589,7.476,148.427
C09799=1196.196,304.924,-69.640,-176.587,7.479,148.427
C09800=1196.192,305.172,-69.669,-176.585,7.482,148.427
C09801=1196.187,305.420,-69.700,-176.582,7.485,148.427
C09802=1196.183,305.668,-69.729,-176.580,7.488,148.427
C09803=1196.179,305.917,-69.760,-176.578,7.490,148.427
C09804=1196.175,306.165,-69.790,-176.575,7.493,148.427
C09805=1196.170,306.413,-69.821,-176.572,7.496,148.427
C09806=1196.166,306.661,-69.851,-176.569,7.499,148.427
C09807=1196.161,306.909,-69.881,-176.567,7.501,148.427
C09808=1196.158,307.157,-69.911,-176.565,7.505,148.427
C09809=1196.153,307.406,-69.941,-176.562,7.508,148.427
C09810=1196.149,307.654,-69.972,-176.560,7.510,148.427
C09811=1196.145,307.902,-70.002,-176.558,7.513,148.427
C09812=1196.141,308.150,-70.032,-176.555,7.516,148.427
C09813=1196.136,308.398,-70.063,-176.552,7.519,148.427
C09814=1196.132,308.646,-70.093,-176.550,7.521,148.427
C09815=1196.127,308.894,-70.124,-176.548,7.524,148.427
C09816=1196.124,309.143,-70.153,-176.545,7.527,148.427
C09817=1196.119,309.391,-70.184,-176.543,7.530,148.427
C09818=1196.115,309.638,-70.214,-176.540,7.533,148.427
C09819=1196.111,309.886,-70.245,-176.538,7.536,148.427
C09820=1196.106,310.135,-70.275,-176.535,7.539,148.427
C09821=1196.103,310.383,-70.306,-176.533,7.541,148.427
C09822=1196.098,310.631,-70.336,-176.530,7.544,148.427
C09823=1196.094,310.879,-70.367,-176.528,7.547,148.427
C09824=1196.089,311.127,-70.397,-176.526,7.551,148.427
C09825=1196.085,311.375,-70.427,-176.523,7.553,148.427
C09826=1196.081,311.624,-70.458,-176.521,7.556,148.427
C09827=1196.077,311.872,-70.489,-176.518,7.559,148.427
C09828=1196.072,312.120,-70.519,-176.516,7.561,148.427
C09829=1196.068,312.367,-70.550,-176.514,7.564,148.427
C09830=1196.064,312.616,-70.581,-176.511,7.567,148.427
C09831=1196.060,312.864,-70.612,-176.508,7.570,148.427
C09832=1196.056,313.112,-70.642,-176.506,7.573,148.427
C09833=1196.051,313.360,-70.672,-176.504,7.576,148.428
C09834=1196.047,313.608,-70.704,-176.501,7.579,148.428
C09835=1196.043,313.856,-70.734,-176.498,7.582,148.428
C09836=1196.039,314.104,-70.765,-176.496,7.584,148.428
C09837=1196.034,314.381,-70.798,-176.493,7.588,148.428
C09838=1196.029,314.657,-70.833,-176.491,7.591,148.428
C09839=1196.025,314.933,-70.867,-176.488,7.594,148.428
C09840=1196.020,315.210,-70.901,-176.485,7.597,148.428
C09841=1196.015,315.458,-70.932,-176.483,7.600,148.428
C09842=1196.011,315.706,-70.963,-176.481,7.604,148.428
C09843=1196.007,315.954,-70.994,-176.478,7.606,148.428
C09844=1196.003,316.202,-71.024,-176.476,7.609,148.428
C09845=1195.999,316.450,-71.056,-176.473,7.612,148.428
C09846=1195.995,316.698,-71.086,-176.471,7.615,148.428
C09847=1195.990,316.946,-71.117,-176.469,7.617,148.428
C09848=1195.986,317.194,-71.148,-176.466,7.620,148.428
C09849=1195.982,317.442,-71.178,-176.464,7.624,148.428
C09850=1195.977,317.690,-71.209,-176.461,7.627,148.428
C09851=1195.973,317.939,-71.240,-176.459,7.629,148.428
C09852=1195.969,318.186,-71.272,-176.457,7.632,148.428
C09853=1195.965,318.434,-71.303,-176.454,7.635,148.428
C09854=1195.961,318.683,-71.334,-176.451,7.638,148.428
C09855=1195.956,318.931,-71.364,-176.450,7.641,148.429
C09856=1195.952,319.178,-71.395,-176.447,7.644,148.429
C09857=1195.948,319.426,-71.426,-176.444,7.647,148.429
C09858=1195.944,319.674,-71.457,-176.442,7.650,148.429
C09859=1195.940,319.923,-71.488,-176.440,7.652,148.429
C09860=1195.935,320.170,-71.520,-176.437,7.655,148.429
C09861=1195.931,320.418,-71.551,-176.435,7.659,148.429
C09862=1195.927,320.667,-71.582,-176.432,7.662,148.429
C09863=1195.922,320.914,-71.613,-176.431,7.664,148.429
C09864=1195.918,321.163,-71.644,-176.428,7.667,148.429
C09865=1195.914,321.411,-71.675,-176.425,7.670,148.429
C09866=1195.910,321.659,-71.707,-176.423,7.674,148.429
C09867=1195.906,321.907,-71.737,-176.421,7.676,148.429
C09868=1195.903,322.155,-71.769,-176.419,7.679,148.429
C09869=1195.898,322.403,-71.800,-176.416,7.682,148.429
C09870=1195.893,322.651,-71.831,-176.413,7.685,148.429
C09871=1195.890,322.899,-71.862,-176.411,7.688,148.430
C09872=1195.885,323.147,-71.893,-176.409,7.691,148.430
C09873=1195.881,323.395,-71.925,-176.407,7.694,148.430
C09874=1195.877,323.643,-71.956,-176.404,7.697,148.430
C09875=1195.873,323.891,-71.988,-176.402,7.700,148.430
C09876=1195.868,324.139,-72.018,-176.399,7.703,148.430
C09877=1195.865,324.387,-72.050,-176.397,7.706,148.430
C09878=1195.860,324.634,-72.081,-176.395,7.709,148.430
C09879=1195.856,324.883,-72.113,-176.392,7.712,148.430
C09880=1195.851,325.131,-72.144,-176.390,7.714,148.430
C09881=1195.847,325.379,-72.176,-176.387,7.717,148.430
C09882=1195.843,325.627,-72.207,-176.385,7.721,148.430
C09883=1195.839,325.875,-72.239,-176.383,7.724,148.430
C09884=1195.835,326.122,-72.270,-176.381,7.726,148.431
C09885=1195.831,326.371,-72.301,-176.378,7.729,148.431
C09886=1195.826,326.618,-72.333,-176.376,7.733,148.431
C09887=1195.822,326.867,-72.364,-176.373,7.736,148.431
C09888=1195.818,327.114,-72.395,-176.372,7.738,148.431
C09889=1195.814,327.363,-72.428,-176.369,7.741,148.431
C09890=1195.810,327.611,-72.459,-176.367,7.745,148.431
C09891=1195.805,327.859,-72.490,-176.364,7.748,148.431
C09892=1195.802,328.107,-72.522,-176.362,7.751,148.431
C09893=1195.797,328.354,-72.554,-176.360,7.753,148.431
C09894=1195.793,328.603,-72.585,-176.357,7.756,148.432
C09895=1195.788,328.850,-72.617,-176.355,7.759,148.432
C09896=1195.784,329.098,-72.649,-176.352,7.763,148.432
C09897=1195.780,329.346,-72.680,-176.350,7.765,148.432
C09898=1195.776,329.594,-72.711,-176.348,7.768,148.432
C09899=1195.772,329.842,-72.743,-176.346,7.772,148.432
C09900=1195.767,330.090,-72.775,-176.343,7.775,148.432
C09901=1195.764,330.338,-72.807,-176.341,7.777,148.432
C09902=1195.759,330.586,-72.838,-176.339,7.780,148.432
C09903=1195.755,330.834,-72.870,-176.337,7.783,148.433
C09904=1195.751,331.082,-72.902,-176.334,7.786,148.433
C09905=1195.747,331.330,-72.934,-176.332,7.790,148.433
C09906=1195.743,331.578,-72.965,-176.330,7.792,148.433
C09907=1195.739,331.825,-72.997,-176.327,7.795,148.433
C09908=1195.734,332.073,-73.029,-176.325,7.799,148.433
C09909=1195.730,332.321,-73.061,-176.323,7.802,148.433
C09910=1195.726,332.569,-73.092,-176.321,7.804,148.433
C09911=1195.721,332.818,-73.124,-176.318,7.808,148.434
C09912=1195.718,333.066,-73.156,-176.316,7.811,148.434
C09913=1195.713,333.313,-73.188,-176.313,7.814,148.434
C09914=1195.709,333.561,-73.220,-176.311,7.817,148.434
C09915=1195.705,333.809,-73.252,-176.309,7.819,148.434
C09916=1195.701,334.057,-73.284,-176.307,7.823,148.434
C09917=1195.697,334.305,-73.316,-176.305,7.826,148.434
C09918=1195.693,334.553,-73.348,-176.302,7.829,148.434
C09919=1195.688,334.801,-73.379,-176.300,7.832,148.435
C09920=1195.684,335.049,-73.412,-176.298,7.835,148.435
C09921=1195.680,335.297,-73.444,-176.296,7.838,148.435
C09922=1195.675,335.545,-73.476,-176.293,7.841,148.435
C09923=1195.672,335.792,-73.508,-176.291,7.845,148.435
C09924=1195.668,336.040,-73.540,-176.289,7.847,148.435
C09925=1195.664,336.288,-73.573,-176.287,7.850,148.435
C09926=1195.659,336.536,-73.604,-176.284,7.853,148.436
C09927=1195.655,336.784,-73.636,-176.282,7.857,148.436
C09928=1195.651,337.032,-73.668,-176.280,7.860,148.436
C09929=1195.646,337.280,-73.700,-176.278,7.862,148.436
C09930=1195.643,337.528,-73.732,-176.275,7.866,148.436
C09931=1195.638,337.776,-73.765,-176.273,7.869,148.436
C09932=1195.635,338.024,-73.797,-176.271,7.872,148.437
C09933=1195.630,338.271,-73.829,-176.269,7.874,148.437
C09934=1195.626,338.519,-73.861,-176.267,7.878,148.437
C09935=1195.622,338.767,-73.894,-176.264,7.881,148.437
C09936=1195.618,339.015,-73.926,-176.262,7.884,148.437
C09937=1195.614,339.263,-73.959,-176.260,7.888,148.438
C09938=1195.609,339.511,-73.990,-176.258,7.890,148.437
C09939=1195.605,339.758,-74.023,-176.256,7.893,148.438
C09940=1195.602,340.006,-74.055,-176.253,7.897,148.438
C09941=1195.597,340.285,-74.092,-176.251,7.900,148.438
C09942=1195.592,340.564,-74.127,-176.249,7.903,148.438
C09943=1195.587,340.842,-74.164,-176.246,7.907,148.438
C09944=1195.583,341.121,-74.200,-176.243,7.910,148.439
C09945=1195.578,341.369,-74.233,-176.241,7.914,148.439
C09946=1195.575,341.616,-74.265,-176.239,7.916,148.439
C09947=1195.570,341.864,-74.297,-176.237,7.920,148.439
C09948=1195.565,342.112,-74.330,-176.235,7.923,148.439
C09949=1195.562,342.360,-74.362,-176.233,7.926,148.440
C09950=1195.558,342.608,-74.395,-176.231,7.930,148.440
C09951=1195.553,342.856,-74.428,-176.229,7.932,148.440
C09952=1195.549,343.103,-74.459,-176.226,7.935,148.440
C09953=1195.545,343.351,-74.493,-176.224,7.938,148.440
C09954=1195.541,343.599,-74.525,-176.222,7.942,148.441
C09955=1195.537,343.847,-74.558,-176.220,7.944,148.441
C09956=1195.533,344.095,-74.590,-176.218,7.948,148.441
C09957=1195.529,344.343,-74.623,-176.216,7.951,148.441
C09958=1195.525,344.591,-74.655,-176.213,7.954,148.441
C09959=1195.520,344.838,-74.688,-176.211,7.958,148.442
C09960=1195.516,345.086,-74.720,-176.209,7.960,148.442
C09961=1195.512,345.334,-74.753,-176.207,7.963,148.442
C09962=1195.508,345.582,-74.785,-176.205,7.967,148.442
C09963=1195.504,345.830,-74.818,-176.203,7.970,148.442
C09964=1195.499,346.078,-74.851,-176.200,7.973,148.443
C09965=1195.496,346.325,-74.883,-176.199,7.976,148.443
C09966=1195.492,346.573,-74.917,-176.197,7.979,148.443
C09967=1195.487,346.821,-74.949,-176.194,7.983,148.443
C09968=1195.483,347.069,-74.982,-176.192,7.986,148.443
C09969=1195.479,347.316,-75.014,-176.190,7.988,148.444
C09970=1195.475,347.564,-75.047,-176.188,7.992,148.444
C09971=1195.471,347.812,-75.080,-176.186,7.995,148.444
C09972=1195.466,348.060,-75.113,-176.184,7.998,148.444
C09973=1195.462,348.308,-75.146,-176.181,8.002,148.445
C09974=1195.459,348.556,-75.178,-176.180,8.005,148.445
C09975=1195.454,348.803,-75.211,-176.178,8.008,148.445
C09976=1195.450,349.051,-75.244,-176.176,8.011,148.445
C09977=1195.446,349.299,-75.277,-176.174,8.015,148.446
C09978=1195.442,349.547,-75.310,-176.172,8.017,148.446
C09979=1195.438,349.795,-75.343,-176.170,8.020,148.446
C09980=1195.434,350.042,-75.376,-176.167,8.024,148.446
C09981=1195.430,350.291,-75.408,-176.165,8.027,148.446
C09982=1195.426,350.538,-75.441,-176.164,8.030,148.447
C09983=1195.421,350.786,-75.474,-176.162,8.033,148.447
C09984=1195.417,351.034,-75.508,-176.159,8.037,148.447
C09985=1195.413,351.282,-75.541,-176.157,8.040,148.448
C09986=1195.409,351.529,-75.574,-176.155,8.043,148.448
C09987=1195.405,351.778,-75.606,-176.154,8.046,148.448
C09988=1195.400,352.025,-75.640,-176.152,8.049,148.448
C09989=1195.397,352.273,-75.672,-176.149,8.053,148.449
C09990=1195.393,352.520,-75.705,-176.147,8.056,148.449
C09991=1195.389,352.768,-75.738,-176.145,8.059,148.449
C09992=1195.385,353.016,-75.772,-176.144,8.062,148.449
C09993=1195.381,353.264,-75.805,-176.141,8.065,148.450
C09994=1195.376,353.511,-75.838,-176.139,8.069,148.450
C09995=1195.372,353.759,-75.871,-176.137,8.072,148.450
C09996=1195.368,354.007,-75.904,-176.136,8.075,148.450
//INST
///DATE 2021/06/15 17:23
///ATTR SC,RW,RJ
////FRAME ROBOT
///GROUP1 RB1
NOP
MOVL C00000 V=800.0 PL=0
MOVL C00001 V=800.0 PL=0
MOVL C00002 V=800.0 PL=0
MOVL C00003 V=800.0 PL=0
MOVL C00004 V=800.0 PL=0
MOVL C00005 V=800.0 PL=0
MOVL C00006 V=800.0 PL=0
MOVL C00007 V=800.0 PL=0
MOVL C00008 V=800.0 PL=0
MOVL C00009 V=800.0 PL=0
MOVL C00010 V=800.0 PL=0
MOVL C00011 V=800.0 PL=0
MOVL C00012 V=800.0 PL=0
MOVL C00013 V=800.0 PL=0
MOVL C00014 V=800.0 PL=0
MOVL C00015 V=800.0 PL=0
MOVL C00016 V=800.0 PL=0
MOVL C00017 V=800.0 PL=0
MOVL C00018 V=800.0 PL=0
MOVL C00019 V=800.0 PL=0
MOVL C00020 V=800.0 PL=0
MOVL C00021 V=800.0 PL=0
MOVL C00022 V=800.0 PL=0
MOVL C00023 V=800.0 PL=0
MOVL C00024 V=800.0 PL=0
MOVL C00025 V=800.0 PL=0
MOVL C00026 V=800.0 PL=0
MOVL C00027 V=800.0 PL=0
MOVL C00028 V=800.0 PL=0
MOVL C00029 V=800.0 PL=0
MOVL C00030 V=800.0 PL=0
MOVL C00031 V=800.0 PL=0
MOVL C00032 V=800.0 PL=0
MOVL C00033 V=800.0 PL=0
MOVL C00034 V=800.0 PL=0
MOVL C00035 V=800.0 PL=0
MOVL C00036 V=800.0 PL=0
MOVL C00037 V=800.0 PL=0
MOVL C00038 V=800.0 PL=0
MOVL C00039 V=800.0 PL=0
MOVL C00040 V=800.0 PL=0
MOVL C00041 V=800.0 PL=0
MOVL C00042 V=800.0 PL=0
MOVL C00043 V=800.0 PL=0
MOVL C00044 V=800.0 PL=0
MOVL C00045 V=800.0 PL=0
MOVL C00046 V=800.0 PL=0
MOVL C00047 V=800.0 PL=0
MOVL C00048 V=800.0 PL=0
MOVL C00049 V=800.0 PL=0
MOVL C00050 V=800.0 PL=0
MOVL C00051 V=800.0 PL=0
MOVL C00052 V=800.0 PL=0
MOVL C00053 V=800.0 PL=0
MOVL C00054 V=800.0 PL=0
MOVL C00055 V=800.0 PL=0
MOVL C00056 V=800.0 PL=0
MOVL C00057 V=800.0 PL=0
MOVL C00058 V=800.0 PL=0
MOVL C00059 V=800.0 PL=0
MOVL C00060 V=800.0 PL=0
MOVL C00061 V=800.0 PL=0
MOVL C00062 V=800.0 PL=0
MOVL C00063 V=800.0 PL=0
MOVL C00064 V=800.0 PL=0
MOVL C00065 V=800.0 PL=0
MOVL C00066 V=800.0 PL=0
MOVL C00067 V=800.0 PL=0
MOVL C00068 V=800.0 PL=0
MOVL C00069 V=800.0 PL=0
MOVL C00070 V=800.0 PL=0
MOVL C00071 V=800.0 PL=0
MOVL C00072 V=800.0 PL=0
MOVL C00073 V=800.0 PL=0
MOVL C00074 V=800.0 PL=0
MOVL C00075 V=800.0 PL=0
MOVL C00076 V=800.0 PL=0
MOVL C00077 V=800.0 PL=0
MOVL C00078 V=800.0 PL=0
MOVL C00079 V=800.0 PL=0
MOVL C00080 V=800.0 PL=0
MOVL C00081 V=800.0 PL=0
MOVL C00082 V=800.0 PL=0
MOVL C00083 V=800.0 PL=0
MOVL C00084 V=800.0 PL=0
MOVL C00085 V=800.0 PL=0
MOVL C00086 V=800.0 PL=0
MOVL C00087 V=800.0 PL=0
MOVL C00088 V=800.0 PL=0
MOVL C00089 V=800.0 PL=0
MOVL C00090 V=800.0 PL=0
MOVL C00091 V=800.0 PL=0
MOVL C00092 V=800.0 PL=0
MOVL C00093 V=800.0 PL=0
MOVL C00094 V=800.0 PL=0
MOVL C00095 V=800.0 PL=0
MOVL C00096 V=800.0 PL=0
MOVL C00097 V=800.0 PL=0
MOVL C00098 V=800.0 PL=0
MOVL C00099 V=800.0 PL=0
MOVL C00100 V=800.0 PL=0
MOVL C00101 V=800.0 PL=0
MOVL C00102 V=800.0 PL=0
MOVL C00103 V=800.0 PL=0
MOVL C00104 V=800.0 PL=0
MOVL C00105 V=800.0 PL=0
MOVL C00106 V=800.0 PL=0
MOVL C00107 V=800.0 PL=0
MOVL C00108 V=800.0 PL=0
MOVL C00109 V=800.0 PL=0
MOVL C00110 V=800.0 PL=0
MOVL C00111 V=800.0 PL=0
MOVL C00112 V=800.0 PL=0
MOVL C00113 V=800.0 PL=0
MOVL C00114 V=800.0 PL=0
MOVL C00115 V=800.0 PL=0
MOVL C00116 V=800.0 PL=0
MOVL C00117 V=800.0 PL=0
MOVL C00118 V=800.0 PL=0
MOVL C00119 V=800.0 PL=0
MOVL C00120 V=800.0 PL=0
MOVL C00121 V=800.0 PL=0
MOVL C00122 V=800.0 PL=0
MOVL C00123 V=800.0 PL=0
MOVL C00124 V=800.0 PL=0
MOVL C00125 V=800.0 PL=0
MOVL C00126 V=800.0 PL=0
MOVL C00127 V=800.0 PL=0
MOVL C00128 V=800.0 PL=0
MOVL C00129 V=800.0 PL=0
MOVL C00130 V=800.0 PL=0
MOVL C00131 V=800.0 PL=0
MOVL C00132 V=800.0 PL=0
MOVL C00133 V=800.0 PL=0
MOVL C00134 V=800.0 PL=0
MOVL C00135 V=800.0 PL=0
MOVL C00136 V=800.0 PL=0
MOVL C00137 V=800.0 PL=0
MOVL C00138 V=800.0 PL=0
MOVL C00139 V=800.0 PL=0
MOVL C00140 V=800.0 PL=0
MOVL C00141 V=800.0 PL=0
MOVL C00142 V=800.0 PL=0
MOVL C00143 V=800.0 PL=0
MOVL C00144 V=800.0 PL=0
MOVL C00145 V=800.0 PL=0
MOVL C00146 V=800.0 PL=0
MOVL C00147 V=800.0 PL=0
MOVL C00148 V=800.0 PL=0
MOVL C00149 V=800.0 PL=0
MOVL C00150 V=800.0 PL=0
MOVL C00151 V=800.0 PL=0
MOVL C00152 V=800.0 PL=0
MOVL C00153 V=800.0 PL=0
MOVL C00154 V=800.0 PL=0
MOVL C00155 V=800.0 PL=0
MOVL C00156 V=800.0 PL=0
MOVL C00157 V=800.0 PL=0
MOVL C00158 V=800.0 PL=0
MOVL C00159 V=800.0 PL=0
MOVL C00160 V=800.0 PL=0
MOVL C00161 V=800.0 PL=0
MOVL C00162 V=800.0 PL=0
MOVL C00163 V=800.0 PL=0
MOVL C00164 V=800.0 PL=0
MOVL C00165 V=800.0 PL=0
MOVL C00166 V=800.0 PL=0
MOVL C00167 V=800.0 PL=0
MOVL C00168 V=800.0 PL=0
MOVL C00169 V=800.0 PL=0
MOVL C00170 V=800.0 PL=0
MOVL C00171 V=800.0 PL=0
MOVL C00172 V=800.0 PL=0
MOVL C00173 V=800.0 PL=0
MOVL C00174 V=800.0 PL=0
MOVL C00175 V=800.0 PL=0
MOVL C00176 V=800.0 PL=0
MOVL C00177 V=800.0 PL=0
MOVL C00178 V=800.0 PL=0
MOVL C00179 V=800.0 PL=0
MOVL C00180 V=800.0 PL=0
MOVL C00181 V=800.0 PL=0
MOVL C00182 V=800.0 PL=0
MOVL C00183 V=800.0 PL=0
MOVL C00184 V=800.0 PL=0
MOVL C00185 V=800.0 PL=0
MOVL C00186 V=800.0 PL=0
MOVL C00187 V=800.0 PL=0
MOVL C00188 V=800.0 PL=0
MOVL C00189 V=800.0 PL=0
MOVL C00190 V=800.0 PL=0
MOVL C00191 V=800.0 PL=0
MOVL C00192 V=800.0 PL=0
MOVL C00193 V=800.0 PL=0
MOVL C00194 V=800.0 PL=0
MOVL C00195 V=800.0 PL=0
MOVL C00196 V=800.0 PL=0
MOVL C00197 V=800.0 PL=0
MOVL C00198 V=800.0 PL=0
MOVL C00199 V=800.0 PL=0
MOVL C00200 V=800.0 PL=0
MOVL C00201 V=800.0 PL=0
MOVL C00202 V=800.0 PL=0
MOVL C00203 V=800.0 PL=0
MOVL C00204 V=800.0 PL=0
MOVL C00205 V=800.0 PL=0
MOVL C00206 V=800.0 PL=0
MOVL C00207 V=800.0 PL=0
MOVL C00208 V=800.0 PL=0
MOVL C00209 V=800.0 PL=0
MOVL C00210 V=800.0 PL=0
MOVL C00211 V=800.0 PL=0
MOVL C00212 V=800.0 PL=0
MOVL C00213 V=800.0 PL=0
MOVL C00214 V=800.0 PL=0
MOVL C00215 V=800.0 PL=0
MOVL C00216 V=800.0 PL=0
MOVL C00217 V=800.0 PL=0
MOVL C00218 V=800.0 PL=0
MOVL C00219 V=800.0 PL=0
MOVL C00220 V=800.0 PL=0
MOVL C00221 V=800.0 PL=0
MOVL C00222 V=800.0 PL=0
MOVL C00223 V=800.0 PL=0
MOVL C00224 V=800.0 PL=0
MOVL C00225 V=800.0 PL=0
MOVL C00226 V=800.0 PL=0
MOVL C00227 V=800.0 PL=0
MOVL C00228 V=800.0 PL=0
MOVL C00229 V=800.0 PL=0
MOVL C00230 V=800.0 PL=0
MOVL C00231 V=800.0 PL=0
MOVL C00232 V=800.0 PL=0
MOVL C00233 V=800.0 PL=0
MOVL C00234 V=800.0 PL=0
MOVL C00235 V=800.0 PL=0
MOVL C00236 V=800.0 PL=0
MOVL C00237 V=800.0 PL=0
MOVL C00238 V=800.0 PL=0
MOVL C00239 V=800.0 PL=0
MOVL C00240 V=800.0 PL=0
MOVL C00241 V=800.0 PL=0
MOVL C00242 V=800.0 PL=0
MOVL C00243 V=800.0 PL=0
MOVL C00244 V=800.0 PL=0
MOVL C00245 V=800.0 PL=0
MOVL C00246 V=800.0 PL=0
MOVL C00247 V=800.0 PL=0
MOVL C00248 V=800.0 PL=0
MOVL C00249 V=800.0 PL=0
MOVL C00250 V=800.0 PL=0
MOVL C00251 V=800.0 PL=0
MOVL C00252 V=800.0 PL=0
MOVL C00253 V=800.0 PL=0
MOVL C00254 V=800.0 PL=0
MOVL C00255 V=800.0 PL=0
MOVL C00256 V=800.0 PL=0
MOVL C00257 V=800.0 PL=0
MOVL C00258 V=800.0 PL=0
MOVL C00259 V=800.0 PL=0
MOVL C00260 V=800.0 PL=0
MOVL C00261 V=800.0 PL=0
MOVL C00262 V=800.0 PL=0
MOVL C00263 V=800.0 PL=0
MOVL C00264 V=800.0 PL=0
MOVL C00265 V=800.0 PL=0
MOVL C00266 V=800.0 PL=0
MOVL C00267 V=800.0 PL=0
MOVL C00268 V=800.0 PL=0
MOVL C00269 V=800.0 PL=0
MOVL C00270 V=800.0 PL=0
MOVL C00271 V=800.0 PL=0
MOVL C00272 V=800.0 PL=0
MOVL C00273 V=800.0 PL=0
MOVL C00274 V=800.0 PL=0
MOVL C00275 V=800.0 PL=0
MOVL C00276 V=800.0 PL=0
MOVL C00277 V=800.0 PL=0
MOVL C00278 V=800.0 PL=0
MOVL C00279 V=800.0 PL=0
MOVL C00280 V=800.0 PL=0
MOVL C00281 V=800.0 PL=0
MOVL C00282 V=800.0 PL=0
MOVL C00283 V=800.0 PL=0
MOVL C00284 V=800.0 PL=0
MOVL C00285 V=800.0 PL=0
MOVL C00286 V=800.0 PL=0
MOVL C00287 V=800.0 PL=0
MOVL C00288 V=800.0 PL=0
MOVL C00289 V=800.0 PL=0
MOVL C00290 V=800.0 PL=0
MOVL C00291 V=800.0 PL=0
MOVL C00292 V=800.0 PL=0
MOVL C00293 V=800.0 PL=0
MOVL C00294 V=800.0 PL=0
MOVL C00295 V=800.0 PL=0
MOVL C00296 V=800.0 PL=0
MOVL C00297 V=800.0 PL=0
MOVL C00298 V=800.0 PL=0
MOVL C00299 V=800.0 PL=0
MOVL C00300 V=800.0 PL=0
MOVL C00301 V=800.0 PL=0
MOVL C00302 V=800.0 PL=0
MOVL C00303 V=800.0 PL=0
MOVL C00304 V=800.0 PL=0
MOVL C00305 V=800.0 PL=0
MOVL C00306 V=800.0 PL=0
MOVL C00307 V=800.0 PL=0
MOVL C00308 V=800.0 PL=0
MOVL C00309 V=800.0 PL=0
MOVL C00310 V=800.0 PL=0
MOVL C00311 V=800.0 PL=0
MOVL C00312 V=800.0 PL=0
MOVL C00313 V=800.0 PL=0
MOVL C00314 V=800.0 PL=0
MOVL C00315 V=800.0 PL=0
MOVL C00316 V=800.0 PL=0
MOVL C00317 V=800.0 PL=0
MOVL C00318 V=800.0 PL=0
MOVL C00319 V=800.0 PL=0
MOVL C00320 V=800.0 PL=0
MOVL C00321 V=800.0 PL=0
MOVL C00322 V=800.0 PL=0
MOVL C00323 V=800.0 PL=0
MOVL C00324 V=800.0 PL=0
MOVL C00325 V=800.0 PL=0
MOVL C00326 V=800.0 PL=0
MOVL C00327 V=800.0 PL=0
MOVL C00328 V=800.0 PL=0
MOVL C00329 V=800.0 PL=0
MOVL C00330 V=800.0 PL=0
MOVL C00331 V=800.0 PL=0
MOVL C00332 V=800.0 PL=0
MOVL C00333 V=800.0 PL=0
MOVL C00334 V=800.0 PL=0
MOVL C00335 V=800.0 PL=0
MOVL C00336 V=800.0 PL=0
MOVL C00337 V=800.0 PL=0
MOVL C00338 V=800.0 PL=0
MOVL C00339 V=800.0 PL=0
MOVL C00340 V=800.0 PL=0
MOVL C00341 V=800.0 PL=0
MOVL C00342 V=800.0 PL=0
MOVL C00343 V=800.0 PL=0
MOVL C00344 V=800.0 PL=0
MOVL C00345 V=800.0 PL=0
MOVL C00346 V=800.0 PL=0
MOVL C00347 V=800.0 PL=0
MOVL C00348 V=800.0 PL=0
MOVL C00349 V=800.0 PL=0
MOVL C00350 V=800.0 PL=0
MOVL C00351 V=800.0 PL=0
MOVL C00352 V=800.0 PL=0
MOVL C00353 V=800.0 PL=0
MOVL C00354 V=800.0 PL=0
MOVL C00355 V=800.0 PL=0
MOVL C00356 V=800.0 PL=0
MOVL C00357 V=800.0 PL=0
MOVL C00358 V=800.0 PL=0
MOVL C00359 V=800.0 PL=0
MOVL C00360 V=800.0 PL=0
MOVL C00361 V=800.0 PL=0
MOVL C00362 V=800.0 PL=0
MOVL C00363 V=800.0 PL=0
MOVL C00364 V=800.0 PL=0
MOVL C00365 V=800.0 PL=0
MOVL C00366 V=800.0 PL=0
MOVL C00367 V=800.0 PL=0
MOVL C00368 V=800.0 PL=0
MOVL C00369 V=800.0 PL=0
MOVL C00370 V=800.0 PL=0
MOVL C00371 V=800.0 PL=0
MOVL C00372 V=800.0 PL=0
MOVL C00373 V=800.0 PL=0
MOVL C00374 V=800.0 PL=0
MOVL C00375 V=800.0 PL=0
MOVL C00376 V=800.0 PL=0
MOVL C00377 V=800.0 PL=0
MOVL C00378 V=800.0 PL=0
MOVL C00379 V=800.0 PL=0
MOVL C00380 V=800.0 PL=0
MOVL C00381 V=800.0 PL=0
MOVL C00382 V=800.0 PL=0
MOVL C00383 V=800.0 PL=0
MOVL C00384 V=800.0 PL=0
MOVL C00385 V=800.0 PL=0
MOVL C00386 V=800.0 PL=0
MOVL C00387 V=800.0 PL=0
MOVL C00388 V=800.0 PL=0
MOVL C00389 V=800.0 PL=0
MOVL C00390 V=800.0 PL=0
MOVL C00391 V=800.0 PL=0
MOVL C00392 V=800.0 PL=0
MOVL C00393 V=800.0 PL=0
MOVL C00394 V=800.0 PL=0
MOVL C00395 V=800.0 PL=0
MOVL C00396 V=800.0 PL=0
MOVL C00397 V=800.0 PL=0
MOVL C00398 V=800.0 PL=0
MOVL C00399 V=800.0 PL=0
MOVL C00400 V=800.0 PL=0
MOVL C00401 V=800.0 PL=0
MOVL C00402 V=800.0 PL=0
MOVL C00403 V=800.0 PL=0
MOVL C00404 V=800.0 PL=0
MOVL C00405 V=800.0 PL=0
MOVL C00406 V=800.0 PL=0
MOVL C00407 V=800.0 PL=0
MOVL C00408 V=800.0 PL=0
MOVL C00409 V=800.0 PL=0
MOVL C00410 V=800.0 PL=0
MOVL C00411 V=800.0 PL=0
MOVL C00412 V=800.0 PL=0
MOVL C00413 V=800.0 PL=0
MOVL C00414 V=800.0 PL=0
MOVL C00415 V=800.0 PL=0
MOVL C00416 V=800.0 PL=0
MOVL C00417 V=800.0 PL=0
MOVL C00418 V=800.0 PL=0
MOVL C00419 V=800.0 PL=0
MOVL C00420 V=800.0 PL=0
MOVL C00421 V=800.0 PL=0
MOVL C00422 V=800.0 PL=0
MOVL C00423 V=800.0 PL=0
MOVL C00424 V=800.0 PL=0
MOVL C00425 V=800.0 PL=0
MOVL C00426 V=800.0 PL=0
MOVL C00427 V=800.0 PL=0
MOVL C00428 V=800.0 PL=0
MOVL C00429 V=800.0 PL=0
MOVL C00430 V=800.0 PL=0
MOVL C00431 V=800.0 PL=0
MOVL C00432 V=800.0 PL=0
MOVL C00433 V=800.0 PL=0
MOVL C00434 V=800.0 PL=0
MOVL C00435 V=800.0 PL=0
MOVL C00436 V=800.0 PL=0
MOVL C00437 V=800.0 PL=0
MOVL C00438 V=800.0 PL=0
MOVL C00439 V=800.0 PL=0
MOVL C00440 V=800.0 PL=0
MOVL C00441 V=800.0 PL=0
MOVL C00442 V=800.0 PL=0
MOVL C00443 V=800.0 PL=0
MOVL C00444 V=800.0 PL=0
MOVL C00445 V=800.0 PL=0
MOVL C00446 V=800.0 PL=0
MOVL C00447 V=800.0 PL=0
MOVL C00448 V=800.0 PL=0
MOVL C00449 V=800.0 PL=0
MOVL C00450 V=800.0 PL=0
MOVL C00451 V=800.0 PL=0
MOVL C00452 V=800.0 PL=0
MOVL C00453 V=800.0 PL=0
MOVL C00454 V=800.0 PL=0
MOVL C00455 V=800.0 PL=0
MOVL C00456 V=800.0 PL=0
MOVL C00457 V=800.0 PL=0
MOVL C00458 V=800.0 PL=0
MOVL C00459 V=800.0 PL=0
MOVL C00460 V=800.0 PL=0
MOVL C00461 V=800.0 PL=0
MOVL C00462 V=800.0 PL=0
MOVL C00463 V=800.0 PL=0
MOVL C00464 V=800.0 PL=0
MOVL C00465 V=800.0 PL=0
MOVL C00466 V=800.0 PL=0
MOVL C00467 V=800.0 PL=0
MOVL C00468 V=800.0 PL=0
MOVL C00469 V=800.0 PL=0
MOVL C00470 V=800.0 PL=0
MOVL C00471 V=800.0 PL=0
MOVL C00472 V=800.0 PL=0
MOVL C00473 V=800.0 PL=0
MOVL C00474 V=800.0 PL=0
MOVL C00475 V=800.0 PL=0
MOVL C00476 V=800.0 PL=0
MOVL C00477 V=800.0 PL=0
MOVL C00478 V=800.0 PL=0
MOVL C00479 V=800.0 PL=0
MOVL C00480 V=800.0 PL=0
MOVL C00481 V=800.0 PL=0
MOVL C00482 V=800.0 PL=0
MOVL C00483 V=800.0 PL=0
MOVL C00484 V=800.0 PL=0
MOVL C00485 V=800.0 PL=0
MOVL C00486 V=800.0 PL=0
MOVL C00487 V=800.0 PL=0
MOVL C00488 V=800.0 PL=0
MOVL C00489 V=800.0 PL=0
MOVL C00490 V=800.0 PL=0
MOVL C00491 V=800.0 PL=0
MOVL C00492 V=800.0 PL=0
MOVL C00493 V=800.0 PL=0
MOVL C00494 V=800.0 PL=0
MOVL C00495 V=800.0 PL=0
MOVL C00496 V=800.0 PL=0
MOVL C00497 V=800.0 PL=0
MOVL C00498 V=800.0 PL=0
MOVL C00499 V=800.0 PL=0
MOVL C00500 V=800.0 PL=0
MOVL C00501 V=800.0 PL=0
MOVL C00502 V=800.0 PL=0
MOVL C00503 V=800.0 PL=0
MOVL C00504 V=800.0 PL=0
MOVL C00505 V=800.0 PL=0
MOVL C00506 V=800.0 PL=0
MOVL C00507 V=800.0 PL=0
MOVL C00508 V=800.0 PL=0
MOVL C00509 V=800.0 PL=0
MOVL C00510 V=800.0 PL=0
MOVL C00511 V=800.0 PL=0
MOVL C00512 V=800.0 PL=0
MOVL C00513 V=800.0 PL=0
MOVL C00514 V=800.0 PL=0
MOVL C00515 V=800.0 PL=0
MOVL C00516 V=800.0 PL=0
MOVL C00517 V=800.0 PL=0
MOVL C00518 V=800.0 PL=0
MOVL C00519 V=800.0 PL=0
MOVL C00520 V=800.0 PL=0
MOVL C00521 V=800.0 PL=0
MOVL C00522 V=800.0 PL=0
MOVL C00523 V=800.0 PL=0
MOVL C00524 V=800.0 PL=0
MOVL C00525 V=800.0 PL=0
MOVL C00526 V=800.0 PL=0
MOVL C00527 V=800.0 PL=0
MOVL C00528 V=800.0 PL=0
MOVL C00529 V=800.0 PL=0
MOVL C00530 V=800.0 PL=0
MOVL C00531 V=800.0 PL=0
MOVL C00532 V=800.0 PL=0
MOVL C00533 V=800.0 PL=0
MOVL C00534 V=800.0 PL=0
MOVL C00535 V=800.0 PL=0
MOVL C00536 V=800.0 PL=0
MOVL C00537 V=800.0 PL=0
MOVL C00538 V=800.0 PL=0
MOVL C00539 V=800.0 PL=0
MOVL C00540 V=800.0 PL=0
MOVL C00541 V=800.0 PL=0
MOVL C00542 V=800.0 PL=0
MOVL C00543 V=800.0 PL=0
MOVL C00544 V=800.0 PL=0
MOVL C00545 V=800.0 PL=0
MOVL C00546 V=800.0 PL=0
MOVL C00547 V=800.0 PL=0
MOVL C00548 V=800.0 PL=0
MOVL C00549 V=800.0 PL=0
MOVL C00550 V=800.0 PL=0
MOVL C00551 V=800.0 PL=0
MOVL C00552 V=800.0 PL=0
MOVL C00553 V=800.0 PL=0
MOVL C00554 V=800.0 PL=0
MOVL C00555 V=800.0 PL=0
MOVL C00556 V=800.0 PL=0
MOVL C00557 V=800.0 PL=0
MOVL C00558 V=800.0 PL=0
MOVL C00559 V=800.0 PL=0
MOVL C00560 V=800.0 PL=0
MOVL C00561 V=800.0 PL=0
MOVL C00562 V=800.0 PL=0
MOVL C00563 V=800.0 PL=0
MOVL C00564 V=800.0 PL=0
MOVL C00565 V=800.0 PL=0
MOVL C00566 V=800.0 PL=0
MOVL C00567 V=800.0 PL=0
MOVL C00568 V=800.0 PL=0
MOVL C00569 V=800.0 PL=0
MOVL C00570 V=800.0 PL=0
MOVL C00571 V=800.0 PL=0
MOVL C00572 V=800.0 PL=0
MOVL C00573 V=800.0 PL=0
MOVL C00574 V=800.0 PL=0
MOVL C00575 V=800.0 PL=0
MOVL C00576 V=800.0 PL=0
MOVL C00577 V=800.0 PL=0
MOVL C00578 V=800.0 PL=0
MOVL C00579 V=800.0 PL=0
MOVL C00580 V=800.0 PL=0
MOVL C00581 V=800.0 PL=0
MOVL C00582 V=800.0 PL=0
MOVL C00583 V=800.0 PL=0
MOVL C00584 V=800.0 PL=0
MOVL C00585 V=800.0 PL=0
MOVL C00586 V=800.0 PL=0
MOVL C00587 V=800.0 PL=0
MOVL C00588 V=800.0 PL=0
MOVL C00589 V=800.0 PL=0
MOVL C00590 V=800.0 PL=0
MOVL C00591 V=800.0 PL=0
MOVL C00592 V=800.0 PL=0
MOVL C00593 V=800.0 PL=0
MOVL C00594 V=800.0 PL=0
MOVL C00595 V=800.0 PL=0
MOVL C00596 V=800.0 PL=0
MOVL C00597 V=800.0 PL=0
MOVL C00598 V=800.0 PL=0
MOVL C00599 V=800.0 PL=0
MOVL C00600 V=800.0 PL=0
MOVL C00601 V=800.0 PL=0
MOVL C00602 V=800.0 PL=0
MOVL C00603 V=800.0 PL=0
MOVL C00604 V=800.0 PL=0
MOVL C00605 V=800.0 PL=0
MOVL C00606 V=800.0 PL=0
MOVL C00607 V=800.0 PL=0
MOVL C00608 V=800.0 PL=0
MOVL C00609 V=800.0 PL=0
MOVL C00610 V=800.0 PL=0
MOVL C00611 V=800.0 PL=0
MOVL C00612 V=800.0 PL=0
MOVL C00613 V=800.0 PL=0
MOVL C00614 V=800.0 PL=0
MOVL C00615 V=800.0 PL=0
MOVL C00616 V=800.0 PL=0
MOVL C00617 V=800.0 PL=0
MOVL C00618 V=800.0 PL=0
MOVL C00619 V=800.0 PL=0
MOVL C00620 V=800.0 PL=0
MOVL C00621 V=800.0 PL=0
MOVL C00622 V=800.0 PL=0
MOVL C00623 V=800.0 PL=0
MOVL C00624 V=800.0 PL=0
MOVL C00625 V=800.0 PL=0
MOVL C00626 V=800.0 PL=0
MOVL C00627 V=800.0 PL=0
MOVL C00628 V=800.0 PL=0
MOVL C00629 V=800.0 PL=0
MOVL C00630 V=800.0 PL=0
MOVL C00631 V=800.0 PL=0
MOVL C00632 V=800.0 PL=0
MOVL C00633 V=800.0 PL=0
MOVL C00634 V=800.0 PL=0
MOVL C00635 V=800.0 PL=0
MOVL C00636 V=800.0 PL=0
MOVL C00637 V=800.0 PL=0
MOVL C00638 V=800.0 PL=0
MOVL C00639 V=800.0 PL=0
MOVL C00640 V=800.0 PL=0
MOVL C00641 V=800.0 PL=0
MOVL C00642 V=800.0 PL=0
MOVL C00643 V=800.0 PL=0
MOVL C00644 V=800.0 PL=0
MOVL C00645 V=800.0 PL=0
MOVL C00646 V=800.0 PL=0
MOVL C00647 V=800.0 PL=0
MOVL C00648 V=800.0 PL=0
MOVL C00649 V=800.0 PL=0
MOVL C00650 V=800.0 PL=0
MOVL C00651 V=800.0 PL=0
MOVL C00652 V=800.0 PL=0
MOVL C00653 V=800.0 PL=0
MOVL C00654 V=800.0 PL=0
MOVL C00655 V=800.0 PL=0
MOVL C00656 V=800.0 PL=0
MOVL C00657 V=800.0 PL=0
MOVL C00658 V=800.0 PL=0
MOVL C00659 V=800.0 PL=0
MOVL C00660 V=800.0 PL=0
MOVL C00661 V=800.0 PL=0
MOVL C00662 V=800.0 PL=0
MOVL C00663 V=800.0 PL=0
MOVL C00664 V=800.0 PL=0
MOVL C00665 V=800.0 PL=0
MOVL C00666 V=800.0 PL=0
MOVL C00667 V=800.0 PL=0
MOVL C00668 V=800.0 PL=0
MOVL C00669 V=800.0 PL=0
MOVL C00670 V=800.0 PL=0
MOVL C00671 V=800.0 PL=0
MOVL C00672 V=800.0 PL=0
MOVL C00673 V=800.0 PL=0
MOVL C00674 V=800.0 PL=0
MOVL C00675 V=800.0 PL=0
MOVL C00676 V=800.0 PL=0
MOVL C00677 V=800.0 PL=0
MOVL C00678 V=800.0 PL=0
MOVL C00679 V=800.0 PL=0
MOVL C00680 V=800.0 PL=0
MOVL C00681 V=800.0 PL=0
MOVL C00682 V=800.0 PL=0
MOVL C00683 V=800.0 PL=0
MOVL C00684 V=800.0 PL=0
MOVL C00685 V=800.0 PL=0
MOVL C00686 V=800.0 PL=0
MOVL C00687 V=800.0 PL=0
MOVL C00688 V=800.0 PL=0
MOVL C00689 V=800.0 PL=0
MOVL C00690 V=800.0 PL=0
MOVL C00691 V=800.0 PL=0
MOVL C00692 V=800.0 PL=0
MOVL C00693 V=800.0 PL=0
MOVL C00694 V=800.0 PL=0
MOVL C00695 V=800.0 PL=0
MOVL C00696 V=800.0 PL=0
MOVL C00697 V=800.0 PL=0
MOVL C00698 V=800.0 PL=0
MOVL C00699 V=800.0 PL=0
MOVL C00700 V=800.0 PL=0
MOVL C00701 V=800.0 PL=0
MOVL C00702 V=800.0 PL=0
MOVL C00703 V=800.0 PL=0
MOVL C00704 V=800.0 PL=0
MOVL C00705 V=800.0 PL=0
MOVL C00706 V=800.0 PL=0
MOVL C00707 V=800.0 PL=0
MOVL C00708 V=800.0 PL=0
MOVL C00709 V=800.0 PL=0
MOVL C00710 V=800.0 PL=0
MOVL C00711 V=800.0 PL=0
MOVL C00712 V=800.0 PL=0
MOVL C00713 V=800.0 PL=0
MOVL C00714 V=800.0 PL=0
MOVL C00715 V=800.0 PL=0
MOVL C00716 V=800.0 PL=0
MOVL C00717 V=800.0 PL=0
MOVL C00718 V=800.0 PL=0
MOVL C00719 V=800.0 PL=0
MOVL C00720 V=800.0 PL=0
MOVL C00721 V=800.0 PL=0
MOVL C00722 V=800.0 PL=0
MOVL C00723 V=800.0 PL=0
MOVL C00724 V=800.0 PL=0
MOVL C00725 V=800.0 PL=0
MOVL C00726 V=800.0 PL=0
MOVL C00727 V=800.0 PL=0
MOVL C00728 V=800.0 PL=0
MOVL C00729 V=800.0 PL=0
MOVL C00730 V=800.0 PL=0
MOVL C00731 V=800.0 PL=0
MOVL C00732 V=800.0 PL=0
MOVL C00733 V=800.0 PL=0
MOVL C00734 V=800.0 PL=0
MOVL C00735 V=800.0 PL=0
MOVL C00736 V=800.0 PL=0
MOVL C00737 V=800.0 PL=0
MOVL C00738 V=800.0 PL=0
MOVL C00739 V=800.0 PL=0
MOVL C00740 V=800.0 PL=0
MOVL C00741 V=800.0 PL=0
MOVL C00742 V=800.0 PL=0
MOVL C00743 V=800.0 PL=0
MOVL C00744 V=800.0 PL=0
MOVL C00745 V=800.0 PL=0
MOVL C00746 V=800.0 PL=0
MOVL C00747 V=800.0 PL=0
MOVL C00748 V=800.0 PL=0
MOVL C00749 V=800.0 PL=0
MOVL C00750 V=800.0 PL=0
MOVL C00751 V=800.0 PL=0
MOVL C00752 V=800.0 PL=0
MOVL C00753 V=800.0 PL=0
MOVL C00754 V=800.0 PL=0
MOVL C00755 V=800.0 PL=0
MOVL C00756 V=800.0 PL=0
MOVL C00757 V=800.0 PL=0
MOVL C00758 V=800.0 PL=0
MOVL C00759 V=800.0 PL=0
MOVL C00760 V=800.0 PL=0
MOVL C00761 V=800.0 PL=0
MOVL C00762 V=800.0 PL=0
MOVL C00763 V=800.0 PL=0
MOVL C00764 V=800.0 PL=0
MOVL C00765 V=800.0 PL=0
MOVL C00766 V=800.0 PL=0
MOVL C00767 V=800.0 PL=0
MOVL C00768 V=800.0 PL=0
MOVL C00769 V=800.0 PL=0
MOVL C00770 V=800.0 PL=0
MOVL C00771 V=800.0 PL=0
MOVL C00772 V=800.0 PL=0
MOVL C00773 V=800.0 PL=0
MOVL C00774 V=800.0 PL=0
MOVL C00775 V=800.0 PL=0
MOVL C00776 V=800.0 PL=0
MOVL C00777 V=800.0 PL=0
MOVL C00778 V=800.0 PL=0
MOVL C00779 V=800.0 PL=0
MOVL C00780 V=800.0 PL=0
MOVL C00781 V=800.0 PL=0
MOVL C00782 V=800.0 PL=0
MOVL C00783 V=800.0 PL=0
MOVL C00784 V=800.0 PL=0
MOVL C00785 V=800.0 PL=0
MOVL C00786 V=800.0 PL=0
MOVL C00787 V=800.0 PL=0
MOVL C00788 V=800.0 PL=0
MOVL C00789 V=800.0 PL=0
MOVL C00790 V=800.0 PL=0
MOVL C00791 V=800.0 PL=0
MOVL C00792 V=800.0 PL=0
MOVL C00793 V=800.0 PL=0
MOVL C00794 V=800.0 PL=0
MOVL C00795 V=800.0 PL=0
MOVL C00796 V=800.0 PL=0
MOVL C00797 V=800.0 PL=0
MOVL C00798 V=800.0 PL=0
MOVL C00799 V=800.0 PL=0
MOVL C00800 V=800.0 PL=0
MOVL C00801 V=800.0 PL=0
MOVL C00802 V=800.0 PL=0
MOVL C00803 V=800.0 PL=0
MOVL C00804 V=800.0 PL=0
MOVL C00805 V=800.0 PL=0
MOVL C00806 V=800.0 PL=0
MOVL C00807 V=800.0 PL=0
MOVL C00808 V=800.0 PL=0
MOVL C00809 V=800.0 PL=0
MOVL C00810 V=800.0 PL=0
MOVL C00811 V=800.0 PL=0
MOVL C00812 V=800.0 PL=0
MOVL C00813 V=800.0 PL=0
MOVL C00814 V=800.0 PL=0
MOVL C00815 V=800.0 PL=0
MOVL C00816 V=800.0 PL=0
MOVL C00817 V=800.0 PL=0
MOVL C00818 V=800.0 PL=0
MOVL C00819 V=800.0 PL=0
MOVL C00820 V=800.0 PL=0
MOVL C00821 V=800.0 PL=0
MOVL C00822 V=800.0 PL=0
MOVL C00823 V=800.0 PL=0
MOVL C00824 V=800.0 PL=0
MOVL C00825 V=800.0 PL=0
MOVL C00826 V=800.0 PL=0
MOVL C00827 V=800.0 PL=0
MOVL C00828 V=800.0 PL=0
MOVL C00829 V=800.0 PL=0
MOVL C00830 V=800.0 PL=0
MOVL C00831 V=800.0 PL=0
MOVL C00832 V=800.0 PL=0
MOVL C00833 V=800.0 PL=0
MOVL C00834 V=800.0 PL=0
MOVL C00835 V=800.0 PL=0
MOVL C00836 V=800.0 PL=0
MOVL C00837 V=800.0 PL=0
MOVL C00838 V=800.0 PL=0
MOVL C00839 V=800.0 PL=0
MOVL C00840 V=800.0 PL=0
MOVL C00841 V=800.0 PL=0
MOVL C00842 V=800.0 PL=0
MOVL C00843 V=800.0 PL=0
MOVL C00844 V=800.0 PL=0
MOVL C00845 V=800.0 PL=0
MOVL C00846 V=800.0 PL=0
MOVL C00847 V=800.0 PL=0
MOVL C00848 V=800.0 PL=0
MOVL C00849 V=800.0 PL=0
MOVL C00850 V=800.0 PL=0
MOVL C00851 V=800.0 PL=0
MOVL C00852 V=800.0 PL=0
MOVL C00853 V=800.0 PL=0
MOVL C00854 V=800.0 PL=0
MOVL C00855 V=800.0 PL=0
MOVL C00856 V=800.0 PL=0
MOVL C00857 V=800.0 PL=0
MOVL C00858 V=800.0 PL=0
MOVL C00859 V=800.0 PL=0
MOVL C00860 V=800.0 PL=0
MOVL C00861 V=800.0 PL=0
MOVL C00862 V=800.0 PL=0
MOVL C00863 V=800.0 PL=0
MOVL C00864 V=800.0 PL=0
MOVL C00865 V=800.0 PL=0
MOVL C00866 V=800.0 PL=0
MOVL C00867 V=800.0 PL=0
MOVL C00868 V=800.0 PL=0
MOVL C00869 V=800.0 PL=0
MOVL C00870 V=800.0 PL=0
MOVL C00871 V=800.0 PL=0
MOVL C00872 V=800.0 PL=0
MOVL C00873 V=800.0 PL=0
MOVL C00874 V=800.0 PL=0
MOVL C00875 V=800.0 PL=0
MOVL C00876 V=800.0 PL=0
MOVL C00877 V=800.0 PL=0
MOVL C00878 V=800.0 PL=0
MOVL C00879 V=800.0 PL=0
MOVL C00880 V=800.0 PL=0
MOVL C00881 V=800.0 PL=0
MOVL C00882 V=800.0 PL=0
MOVL C00883 V=800.0 PL=0
MOVL C00884 V=800.0 PL=0
MOVL C00885 V=800.0 PL=0
MOVL C00886 V=800.0 PL=0
MOVL C00887 V=800.0 PL=0
MOVL C00888 V=800.0 PL=0
MOVL C00889 V=800.0 PL=0
MOVL C00890 V=800.0 PL=0
MOVL C00891 V=800.0 PL=0
MOVL C00892 V=800.0 PL=0
MOVL C00893 V=800.0 PL=0
MOVL C00894 V=800.0 PL=0
MOVL C00895 V=800.0 PL=0
MOVL C00896 V=800.0 PL=0
MOVL C00897 V=800.0 PL=0
MOVL C00898 V=800.0 PL=0
MOVL C00899 V=800.0 PL=0
MOVL C00900 V=800.0 PL=0
MOVL C00901 V=800.0 PL=0
MOVL C00902 V=800.0 PL=0
MOVL C00903 V=800.0 PL=0
MOVL C00904 V=800.0 PL=0
MOVL C00905 V=800.0 PL=0
MOVL C00906 V=800.0 PL=0
MOVL C00907 V=800.0 PL=0
MOVL C00908 V=800.0 PL=0
MOVL C00909 V=800.0 PL=0
MOVL C00910 V=800.0 PL=0
MOVL C00911 V=800.0 PL=0
MOVL C00912 V=800.0 PL=0
MOVL C00913 V=800.0 PL=0
MOVL C00914 V=800.0 PL=0
MOVL C00915 V=800.0 PL=0
MOVL C00916 V=800.0 PL=0
MOVL C00917 V=800.0 PL=0
MOVL C00918 V=800.0 PL=0
MOVL C00919 V=800.0 PL=0
MOVL C00920 V=800.0 PL=0
MOVL C00921 V=800.0 PL=0
MOVL C00922 V=800.0 PL=0
MOVL C00923 V=800.0 PL=0
MOVL C00924 V=800.0 PL=0
MOVL C00925 V=800.0 PL=0
MOVL C00926 V=800.0 PL=0
MOVL C00927 V=800.0 PL=0
MOVL C00928 V=800.0 PL=0
MOVL C00929 V=800.0 PL=0
MOVL C00930 V=800.0 PL=0
MOVL C00931 V=800.0 PL=0
MOVL C00932 V=800.0 PL=0
MOVL C00933 V=800.0 PL=0
MOVL C00934 V=800.0 PL=0
MOVL C00935 V=800.0 PL=0
MOVL C00936 V=800.0 PL=0
MOVL C00937 V=800.0 PL=0
MOVL C00938 V=800.0 PL=0
MOVL C00939 V=800.0 PL=0
MOVL C00940 V=800.0 PL=0
MOVL C00941 V=800.0 PL=0
MOVL C00942 V=800.0 PL=0
MOVL C00943 V=800.0 PL=0
MOVL C00944 V=800.0 PL=0
MOVL C00945 V=800.0 PL=0
MOVL C00946 V=800.0 PL=0
MOVL C00947 V=800.0 PL=0
MOVL C00948 V=800.0 PL=0
MOVL C00949 V=800.0 PL=0
MOVL C00950 V=800.0 PL=0
MOVL C00951 V=800.0 PL=0
MOVL C00952 V=800.0 PL=0
MOVL C00953 V=800.0 PL=0
MOVL C00954 V=800.0 PL=0
MOVL C00955 V=800.0 PL=0
MOVL C00956 V=800.0 PL=0
MOVL C00957 V=800.0 PL=0
MOVL C00958 V=800.0 PL=0
MOVL C00959 V=800.0 PL=0
MOVL C00960 V=800.0 PL=0
MOVL C00961 V=800.0 PL=0
MOVL C00962 V=800.0 PL=0
MOVL C00963 V=800.0 PL=0
MOVL C00964 V=800.0 PL=0
MOVL C00965 V=800.0 PL=0
MOVL C00966 V=800.0 PL=0
MOVL C00967 V=800.0 PL=0
MOVL C00968 V=800.0 PL=0
MOVL C00969 V=800.0 PL=0
MOVL C00970 V=800.0 PL=0
MOVL C00971 V=800.0 PL=0
MOVL C00972 V=800.0 PL=0
MOVL C00973 V=800.0 PL=0
MOVL C00974 V=800.0 PL=0
MOVL C00975 V=800.0 PL=0
MOVL C00976 V=800.0 PL=0
MOVL C00977 V=800.0 PL=0
MOVL C00978 V=800.0 PL=0
MOVL C00979 V=800.0 PL=0
MOVL C00980 V=800.0 PL=0
MOVL C00981 V=800.0 PL=0
MOVL C00982 V=800.0 PL=0
MOVL C00983 V=800.0 PL=0
MOVL C00984 V=800.0 PL=0
MOVL C00985 V=800.0 PL=0
MOVL C00986 V=800.0 PL=0
MOVL C00987 V=800.0 PL=0
MOVL C00988 V=800.0 PL=0
MOVL C00989 V=800.0 PL=0
MOVL C00990 V=800.0 PL=0
MOVL C00991 V=800.0 PL=0
MOVL C00992 V=800.0 PL=0
MOVL C00993 V=800.0 PL=0
MOVL C00994 V=800.0 PL=0
MOVL C00995 V=800.0 PL=0
MOVL C00996 V=800.0 PL=0
MOVL C00997 V=800.0 PL=0
MOVL C00998 V=800.0 PL=0
MOVL C00999 V=800.0 PL=0
MOVL C01000 V=800.0 PL=0
MOVL C01001 V=800.0 PL=0
MOVL C01002 V=800.0 PL=0
MOVL C01003 V=800.0 PL=0
MOVL C01004 V=800.0 PL=0
MOVL C01005 V=800.0 PL=0
MOVL C01006 V=800.0 PL=0
MOVL C01007 V=800.0 PL=0
MOVL C01008 V=800.0 PL=0
MOVL C01009 V=800.0 PL=0
MOVL C01010 V=800.0 PL=0
MOVL C01011 V=800.0 PL=0
MOVL C01012 V=800.0 PL=0
MOVL C01013 V=800.0 PL=0
MOVL C01014 V=800.0 PL=0
MOVL C01015 V=800.0 PL=0
MOVL C01016 V=800.0 PL=0
MOVL C01017 V=800.0 PL=0
MOVL C01018 V=800.0 PL=0
MOVL C01019 V=800.0 PL=0
MOVL C01020 V=800.0 PL=0
MOVL C01021 V=800.0 PL=0
MOVL C01022 V=800.0 PL=0
MOVL C01023 V=800.0 PL=0
MOVL C01024 V=800.0 PL=0
MOVL C01025 V=800.0 PL=0
MOVL C01026 V=800.0 PL=0
MOVL C01027 V=800.0 PL=0
MOVL C01028 V=800.0 PL=0
MOVL C01029 V=800.0 PL=0
MOVL C01030 V=800.0 PL=0
MOVL C01031 V=800.0 PL=0
MOVL C01032 V=800.0 PL=0
MOVL C01033 V=800.0 PL=0
MOVL C01034 V=800.0 PL=0
MOVL C01035 V=800.0 PL=0
MOVL C01036 V=800.0 PL=0
MOVL C01037 V=800.0 PL=0
MOVL C01038 V=800.0 PL=0
MOVL C01039 V=800.0 PL=0
MOVL C01040 V=800.0 PL=0
MOVL C01041 V=800.0 PL=0
MOVL C01042 V=800.0 PL=0
MOVL C01043 V=800.0 PL=0
MOVL C01044 V=800.0 PL=0
MOVL C01045 V=800.0 PL=0
MOVL C01046 V=800.0 PL=0
MOVL C01047 V=800.0 PL=0
MOVL C01048 V=800.0 PL=0
MOVL C01049 V=800.0 PL=0
MOVL C01050 V=800.0 PL=0
MOVL C01051 V=800.0 PL=0
MOVL C01052 V=800.0 PL=0
MOVL C01053 V=800.0 PL=0
MOVL C01054 V=800.0 PL=0
MOVL C01055 V=800.0 PL=0
MOVL C01056 V=800.0 PL=0
MOVL C01057 V=800.0 PL=0
MOVL C01058 V=800.0 PL=0
MOVL C01059 V=800.0 PL=0
MOVL C01060 V=800.0 PL=0
MOVL C01061 V=800.0 PL=0
MOVL C01062 V=800.0 PL=0
MOVL C01063 V=800.0 PL=0
MOVL C01064 V=800.0 PL=0
MOVL C01065 V=800.0 PL=0
MOVL C01066 V=800.0 PL=0
MOVL C01067 V=800.0 PL=0
MOVL C01068 V=800.0 PL=0
MOVL C01069 V=800.0 PL=0
MOVL C01070 V=800.0 PL=0
MOVL C01071 V=800.0 PL=0
MOVL C01072 V=800.0 PL=0
MOVL C01073 V=800.0 PL=0
MOVL C01074 V=800.0 PL=0
MOVL C01075 V=800.0 PL=0
MOVL C01076 V=800.0 PL=0
MOVL C01077 V=800.0 PL=0
MOVL C01078 V=800.0 PL=0
MOVL C01079 V=800.0 PL=0
MOVL C01080 V=800.0 PL=0
MOVL C01081 V=800.0 PL=0
MOVL C01082 V=800.0 PL=0
MOVL C01083 V=800.0 PL=0
MOVL C01084 V=800.0 PL=0
MOVL C01085 V=800.0 PL=0
MOVL C01086 V=800.0 PL=0
MOVL C01087 V=800.0 PL=0
MOVL C01088 V=800.0 PL=0
MOVL C01089 V=800.0 PL=0
MOVL C01090 V=800.0 PL=0
MOVL C01091 V=800.0 PL=0
MOVL C01092 V=800.0 PL=0
MOVL C01093 V=800.0 PL=0
MOVL C01094 V=800.0 PL=0
MOVL C01095 V=800.0 PL=0
MOVL C01096 V=800.0 PL=0
MOVL C01097 V=800.0 PL=0
MOVL C01098 V=800.0 PL=0
MOVL C01099 V=800.0 PL=0
MOVL C01100 V=800.0 PL=0
MOVL C01101 V=800.0 PL=0
MOVL C01102 V=800.0 PL=0
MOVL C01103 V=800.0 PL=0
MOVL C01104 V=800.0 PL=0
MOVL C01105 V=800.0 PL=0
MOVL C01106 V=800.0 PL=0
MOVL C01107 V=800.0 PL=0
MOVL C01108 V=800.0 PL=0
MOVL C01109 V=800.0 PL=0
MOVL C01110 V=800.0 PL=0
MOVL C01111 V=800.0 PL=0
MOVL C01112 V=800.0 PL=0
MOVL C01113 V=800.0 PL=0
MOVL C01114 V=800.0 PL=0
MOVL C01115 V=800.0 PL=0
MOVL C01116 V=800.0 PL=0
MOVL C01117 V=800.0 PL=0
MOVL C01118 V=800.0 PL=0
MOVL C01119 V=800.0 PL=0
MOVL C01120 V=800.0 PL=0
MOVL C01121 V=800.0 PL=0
MOVL C01122 V=800.0 PL=0
MOVL C01123 V=800.0 PL=0
MOVL C01124 V=800.0 PL=0
MOVL C01125 V=800.0 PL=0
MOVL C01126 V=800.0 PL=0
MOVL C01127 V=800.0 PL=0
MOVL C01128 V=800.0 PL=0
MOVL C01129 V=800.0 PL=0
MOVL C01130 V=800.0 PL=0
MOVL C01131 V=800.0 PL=0
MOVL C01132 V=800.0 PL=0
MOVL C01133 V=800.0 PL=0
MOVL C01134 V=800.0 PL=0
MOVL C01135 V=800.0 PL=0
MOVL C01136 V=800.0 PL=0
MOVL C01137 V=800.0 PL=0
MOVL C01138 V=800.0 PL=0
MOVL C01139 V=800.0 PL=0
MOVL C01140 V=800.0 PL=0
MOVL C01141 V=800.0 PL=0
MOVL C01142 V=800.0 PL=0
MOVL C01143 V=800.0 PL=0
MOVL C01144 V=800.0 PL=0
MOVL C01145 V=800.0 PL=0
MOVL C01146 V=800.0 PL=0
MOVL C01147 V=800.0 PL=0
MOVL C01148 V=800.0 PL=0
MOVL C01149 V=800.0 PL=0
MOVL C01150 V=800.0 PL=0
MOVL C01151 V=800.0 PL=0
MOVL C01152 V=800.0 PL=0
MOVL C01153 V=800.0 PL=0
MOVL C01154 V=800.0 PL=0
MOVL C01155 V=800.0 PL=0
MOVL C01156 V=800.0 PL=0
MOVL C01157 V=800.0 PL=0
MOVL C01158 V=800.0 PL=0
MOVL C01159 V=800.0 PL=0
MOVL C01160 V=800.0 PL=0
MOVL C01161 V=800.0 PL=0
MOVL C01162 V=800.0 PL=0
MOVL C01163 V=800.0 PL=0
MOVL C01164 V=800.0 PL=0
MOVL C01165 V=800.0 PL=0
MOVL C01166 V=800.0 PL=0
MOVL C01167 V=800.0 PL=0
MOVL C01168 V=800.0 PL=0
MOVL C01169 V=800.0 PL=0
MOVL C01170 V=800.0 PL=0
MOVL C01171 V=800.0 PL=0
MOVL C01172 V=800.0 PL=0
MOVL C01173 V=800.0 PL=0
MOVL C01174 V=800.0 PL=0
MOVL C01175 V=800.0 PL=0
MOVL C01176 V=800.0 PL=0
MOVL C01177 V=800.0 PL=0
MOVL C01178 V=800.0 PL=0
MOVL C01179 V=800.0 PL=0
MOVL C01180 V=800.0 PL=0
MOVL C01181 V=800.0 PL=0
MOVL C01182 V=800.0 PL=0
MOVL C01183 V=800.0 PL=0
MOVL C01184 V=800.0 PL=0
MOVL C01185 V=800.0 PL=0
MOVL C01186 V=800.0 PL=0
MOVL C01187 V=800.0 PL=0
MOVL C01188 V=800.0 PL=0
MOVL C01189 V=800.0 PL=0
MOVL C01190 V=800.0 PL=0
MOVL C01191 V=800.0 PL=0
MOVL C01192 V=800.0 PL=0
MOVL C01193 V=800.0 PL=0
MOVL C01194 V=800.0 PL=0
MOVL C01195 V=800.0 PL=0
MOVL C01196 V=800.0 PL=0
MOVL C01197 V=800.0 PL=0
MOVL C01198 V=800.0 PL=0
MOVL C01199 V=800.0 PL=0
MOVL C01200 V=800.0 PL=0
MOVL C01201 V=800.0 PL=0
MOVL C01202 V=800.0 PL=0
MOVL C01203 V=800.0 PL=0
MOVL C01204 V=800.0 PL=0
MOVL C01205 V=800.0 PL=0
MOVL C01206 V=800.0 PL=0
MOVL C01207 V=800.0 PL=0
MOVL C01208 V=800.0 PL=0
MOVL C01209 V=800.0 PL=0
MOVL C01210 V=800.0 PL=0
MOVL C01211 V=800.0 PL=0
MOVL C01212 V=800.0 PL=0
MOVL C01213 V=800.0 PL=0
MOVL C01214 V=800.0 PL=0
MOVL C01215 V=800.0 PL=0
MOVL C01216 V=800.0 PL=0
MOVL C01217 V=800.0 PL=0
MOVL C01218 V=800.0 PL=0
MOVL C01219 V=800.0 PL=0
MOVL C01220 V=800.0 PL=0
MOVL C01221 V=800.0 PL=0
MOVL C01222 V=800.0 PL=0
MOVL C01223 V=800.0 PL=0
MOVL C01224 V=800.0 PL=0
MOVL C01225 V=800.0 PL=0
MOVL C01226 V=800.0 PL=0
MOVL C01227 V=800.0 PL=0
MOVL C01228 V=800.0 PL=0
MOVL C01229 V=800.0 PL=0
MOVL C01230 V=800.0 PL=0
MOVL C01231 V=800.0 PL=0
MOVL C01232 V=800.0 PL=0
MOVL C01233 V=800.0 PL=0
MOVL C01234 V=800.0 PL=0
MOVL C01235 V=800.0 PL=0
MOVL C01236 V=800.0 PL=0
MOVL C01237 V=800.0 PL=0
MOVL C01238 V=800.0 PL=0
MOVL C01239 V=800.0 PL=0
MOVL C01240 V=800.0 PL=0
MOVL C01241 V=800.0 PL=0
MOVL C01242 V=800.0 PL=0
MOVL C01243 V=800.0 PL=0
MOVL C01244 V=800.0 PL=0
MOVL C01245 V=800.0 PL=0
MOVL C01246 V=800.0 PL=0
MOVL C01247 V=800.0 PL=0
MOVL C01248 V=800.0 PL=0
MOVL C01249 V=800.0 PL=0
MOVL C01250 V=800.0 PL=0
MOVL C01251 V=800.0 PL=0
MOVL C01252 V=800.0 PL=0
MOVL C01253 V=800.0 PL=0
MOVL C01254 V=800.0 PL=0
MOVL C01255 V=800.0 PL=0
MOVL C01256 V=800.0 PL=0
MOVL C01257 V=800.0 PL=0
MOVL C01258 V=800.0 PL=0
MOVL C01259 V=800.0 PL=0
MOVL C01260 V=800.0 PL=0
MOVL C01261 V=800.0 PL=0
MOVL C01262 V=800.0 PL=0
MOVL C01263 V=800.0 PL=0
MOVL C01264 V=800.0 PL=0
MOVL C01265 V=800.0 PL=0
MOVL C01266 V=800.0 PL=0
MOVL C01267 V=800.0 PL=0
MOVL C01268 V=800.0 PL=0
MOVL C01269 V=800.0 PL=0
MOVL C01270 V=800.0 PL=0
MOVL C01271 V=800.0 PL=0
MOVL C01272 V=800.0 PL=0
MOVL C01273 V=800.0 PL=0
MOVL C01274 V=800.0 PL=0
MOVL C01275 V=800.0 PL=0
MOVL C01276 V=800.0 PL=0
MOVL C01277 V=800.0 PL=0
MOVL C01278 V=800.0 PL=0
MOVL C01279 V=800.0 PL=0
MOVL C01280 V=800.0 PL=0
MOVL C01281 V=800.0 PL=0
MOVL C01282 V=800.0 PL=0
MOVL C01283 V=800.0 PL=0
MOVL C01284 V=800.0 PL=0
MOVL C01285 V=800.0 PL=0
MOVL C01286 V=800.0 PL=0
MOVL C01287 V=800.0 PL=0
MOVL C01288 V=800.0 PL=0
MOVL C01289 V=800.0 PL=0
MOVL C01290 V=800.0 PL=0
MOVL C01291 V=800.0 PL=0
MOVL C01292 V=800.0 PL=0
MOVL C01293 V=800.0 PL=0
MOVL C01294 V=800.0 PL=0
MOVL C01295 V=800.0 PL=0
MOVL C01296 V=800.0 PL=0
MOVL C01297 V=800.0 PL=0
MOVL C01298 V=800.0 PL=0
MOVL C01299 V=800.0 PL=0
MOVL C01300 V=800.0 PL=0
MOVL C01301 V=800.0 PL=0
MOVL C01302 V=800.0 PL=0
MOVL C01303 V=800.0 PL=0
MOVL C01304 V=800.0 PL=0
MOVL C01305 V=800.0 PL=0
MOVL C01306 V=800.0 PL=0
MOVL C01307 V=800.0 PL=0
MOVL C01308 V=800.0 PL=0
MOVL C01309 V=800.0 PL=0
MOVL C01310 V=800.0 PL=0
MOVL C01311 V=800.0 PL=0
MOVL C01312 V=800.0 PL=0
MOVL C01313 V=800.0 PL=0
MOVL C01314 V=800.0 PL=0
MOVL C01315 V=800.0 PL=0
MOVL C01316 V=800.0 PL=0
MOVL C01317 V=800.0 PL=0
MOVL C01318 V=800.0 PL=0
MOVL C01319 V=800.0 PL=0
MOVL C01320 V=800.0 PL=0
MOVL C01321 V=800.0 PL=0
MOVL C01322 V=800.0 PL=0
MOVL C01323 V=800.0 PL=0
MOVL C01324 V=800.0 PL=0
MOVL C01325 V=800.0 PL=0
MOVL C01326 V=800.0 PL=0
MOVL C01327 V=800.0 PL=0
MOVL C01328 V=800.0 PL=0
MOVL C01329 V=800.0 PL=0
MOVL C01330 V=800.0 PL=0
MOVL C01331 V=800.0 PL=0
MOVL C01332 V=800.0 PL=0
MOVL C01333 V=800.0 PL=0
MOVL C01334 V=800.0 PL=0
MOVL C01335 V=800.0 PL=0
MOVL C01336 V=800.0 PL=0
MOVL C01337 V=800.0 PL=0
MOVL C01338 V=800.0 PL=0
MOVL C01339 V=800.0 PL=0
MOVL C01340 V=800.0 PL=0
MOVL C01341 V=800.0 PL=0
MOVL C01342 V=800.0 PL=0
MOVL C01343 V=800.0 PL=0
MOVL C01344 V=800.0 PL=0
MOVL C01345 V=800.0 PL=0
MOVL C01346 V=800.0 PL=0
MOVL C01347 V=800.0 PL=0
MOVL C01348 V=800.0 PL=0
MOVL C01349 V=800.0 PL=0
MOVL C01350 V=800.0 PL=0
MOVL C01351 V=800.0 PL=0
MOVL C01352 V=800.0 PL=0
MOVL C01353 V=800.0 PL=0
MOVL C01354 V=800.0 PL=0
MOVL C01355 V=800.0 PL=0
MOVL C01356 V=800.0 PL=0
MOVL C01357 V=800.0 PL=0
MOVL C01358 V=800.0 PL=0
MOVL C01359 V=800.0 PL=0
MOVL C01360 V=800.0 PL=0
MOVL C01361 V=800.0 PL=0
MOVL C01362 V=800.0 PL=0
MOVL C01363 V=800.0 PL=0
MOVL C01364 V=800.0 PL=0
MOVL C01365 V=800.0 PL=0
MOVL C01366 V=800.0 PL=0
MOVL C01367 V=800.0 PL=0
MOVL C01368 V=800.0 PL=0
MOVL C01369 V=800.0 PL=0
MOVL C01370 V=800.0 PL=0
MOVL C01371 V=800.0 PL=0
MOVL C01372 V=800.0 PL=0
MOVL C01373 V=800.0 PL=0
MOVL C01374 V=800.0 PL=0
MOVL C01375 V=800.0 PL=0
MOVL C01376 V=800.0 PL=0
MOVL C01377 V=800.0 PL=0
MOVL C01378 V=800.0 PL=0
MOVL C01379 V=800.0 PL=0
MOVL C01380 V=800.0 PL=0
MOVL C01381 V=800.0 PL=0
MOVL C01382 V=800.0 PL=0
MOVL C01383 V=800.0 PL=0
MOVL C01384 V=800.0 PL=0
MOVL C01385 V=800.0 PL=0
MOVL C01386 V=800.0 PL=0
MOVL C01387 V=800.0 PL=0
MOVL C01388 V=800.0 PL=0
MOVL C01389 V=800.0 PL=0
MOVL C01390 V=800.0 PL=0
MOVL C01391 V=800.0 PL=0
MOVL C01392 V=800.0 PL=0
MOVL C01393 V=800.0 PL=0
MOVL C01394 V=800.0 PL=0
MOVL C01395 V=800.0 PL=0
MOVL C01396 V=800.0 PL=0
MOVL C01397 V=800.0 PL=0
MOVL C01398 V=800.0 PL=0
MOVL C01399 V=800.0 PL=0
MOVL C01400 V=800.0 PL=0
MOVL C01401 V=800.0 PL=0
MOVL C01402 V=800.0 PL=0
MOVL C01403 V=800.0 PL=0
MOVL C01404 V=800.0 PL=0
MOVL C01405 V=800.0 PL=0
MOVL C01406 V=800.0 PL=0
MOVL C01407 V=800.0 PL=0
MOVL C01408 V=800.0 PL=0
MOVL C01409 V=800.0 PL=0
MOVL C01410 V=800.0 PL=0
MOVL C01411 V=800.0 PL=0
MOVL C01412 V=800.0 PL=0
MOVL C01413 V=800.0 PL=0
MOVL C01414 V=800.0 PL=0
MOVL C01415 V=800.0 PL=0
MOVL C01416 V=800.0 PL=0
MOVL C01417 V=800.0 PL=0
MOVL C01418 V=800.0 PL=0
MOVL C01419 V=800.0 PL=0
MOVL C01420 V=800.0 PL=0
MOVL C01421 V=800.0 PL=0
MOVL C01422 V=800.0 PL=0
MOVL C01423 V=800.0 PL=0
MOVL C01424 V=800.0 PL=0
MOVL C01425 V=800.0 PL=0
MOVL C01426 V=800.0 PL=0
MOVL C01427 V=800.0 PL=0
MOVL C01428 V=800.0 PL=0
MOVL C01429 V=800.0 PL=0
MOVL C01430 V=800.0 PL=0
MOVL C01431 V=800.0 PL=0
MOVL C01432 V=800.0 PL=0
MOVL C01433 V=800.0 PL=0
MOVL C01434 V=800.0 PL=0
MOVL C01435 V=800.0 PL=0
MOVL C01436 V=800.0 PL=0
MOVL C01437 V=800.0 PL=0
MOVL C01438 V=800.0 PL=0
MOVL C01439 V=800.0 PL=0
MOVL C01440 V=800.0 PL=0
MOVL C01441 V=800.0 PL=0
MOVL C01442 V=800.0 PL=0
MOVL C01443 V=800.0 PL=0
MOVL C01444 V=800.0 PL=0
MOVL C01445 V=800.0 PL=0
MOVL C01446 V=800.0 PL=0
MOVL C01447 V=800.0 PL=0
MOVL C01448 V=800.0 PL=0
MOVL C01449 V=800.0 PL=0
MOVL C01450 V=800.0 PL=0
MOVL C01451 V=800.0 PL=0
MOVL C01452 V=800.0 PL=0
MOVL C01453 V=800.0 PL=0
MOVL C01454 V=800.0 PL=0
MOVL C01455 V=800.0 PL=0
MOVL C01456 V=800.0 PL=0
MOVL C01457 V=800.0 PL=0
MOVL C01458 V=800.0 PL=0
MOVL C01459 V=800.0 PL=0
MOVL C01460 V=800.0 PL=0
MOVL C01461 V=800.0 PL=0
MOVL C01462 V=800.0 PL=0
MOVL C01463 V=800.0 PL=0
MOVL C01464 V=800.0 PL=0
MOVL C01465 V=800.0 PL=0
MOVL C01466 V=800.0 PL=0
MOVL C01467 V=800.0 PL=0
MOVL C01468 V=800.0 PL=0
MOVL C01469 V=800.0 PL=0
MOVL C01470 V=800.0 PL=0
MOVL C01471 V=800.0 PL=0
MOVL C01472 V=800.0 PL=0
MOVL C01473 V=800.0 PL=0
MOVL C01474 V=800.0 PL=0
MOVL C01475 V=800.0 PL=0
MOVL C01476 V=800.0 PL=0
MOVL C01477 V=800.0 PL=0
MOVL C01478 V=800.0 PL=0
MOVL C01479 V=800.0 PL=0
MOVL C01480 V=800.0 PL=0
MOVL C01481 V=800.0 PL=0
MOVL C01482 V=800.0 PL=0
MOVL C01483 V=800.0 PL=0
MOVL C01484 V=800.0 PL=0
MOVL C01485 V=800.0 PL=0
MOVL C01486 V=800.0 PL=0
MOVL C01487 V=800.0 PL=0
MOVL C01488 V=800.0 PL=0
MOVL C01489 V=800.0 PL=0
MOVL C01490 V=800.0 PL=0
MOVL C01491 V=800.0 PL=0
MOVL C01492 V=800.0 PL=0
MOVL C01493 V=800.0 PL=0
MOVL C01494 V=800.0 PL=0
MOVL C01495 V=800.0 PL=0
MOVL C01496 V=800.0 PL=0
MOVL C01497 V=800.0 PL=0
MOVL C01498 V=800.0 PL=0
MOVL C01499 V=800.0 PL=0
MOVL C01500 V=800.0 PL=0
MOVL C01501 V=800.0 PL=0
MOVL C01502 V=800.0 PL=0
MOVL C01503 V=800.0 PL=0
MOVL C01504 V=800.0 PL=0
MOVL C01505 V=800.0 PL=0
MOVL C01506 V=800.0 PL=0
MOVL C01507 V=800.0 PL=0
MOVL C01508 V=800.0 PL=0
MOVL C01509 V=800.0 PL=0
MOVL C01510 V=800.0 PL=0
MOVL C01511 V=800.0 PL=0
MOVL C01512 V=800.0 PL=0
MOVL C01513 V=800.0 PL=0
MOVL C01514 V=800.0 PL=0
MOVL C01515 V=800.0 PL=0
MOVL C01516 V=800.0 PL=0
MOVL C01517 V=800.0 PL=0
MOVL C01518 V=800.0 PL=0
MOVL C01519 V=800.0 PL=0
MOVL C01520 V=800.0 PL=0
MOVL C01521 V=800.0 PL=0
MOVL C01522 V=800.0 PL=0
MOVL C01523 V=800.0 PL=0
MOVL C01524 V=800.0 PL=0
MOVL C01525 V=800.0 PL=0
MOVL C01526 V=800.0 PL=0
MOVL C01527 V=800.0 PL=0
MOVL C01528 V=800.0 PL=0
MOVL C01529 V=800.0 PL=0
MOVL C01530 V=800.0 PL=0
MOVL C01531 V=800.0 PL=0
MOVL C01532 V=800.0 PL=0
MOVL C01533 V=800.0 PL=0
MOVL C01534 V=800.0 PL=0
MOVL C01535 V=800.0 PL=0
MOVL C01536 V=800.0 PL=0
MOVL C01537 V=800.0 PL=0
MOVL C01538 V=800.0 PL=0
MOVL C01539 V=800.0 PL=0
MOVL C01540 V=800.0 PL=0
MOVL C01541 V=800.0 PL=0
MOVL C01542 V=800.0 PL=0
MOVL C01543 V=800.0 PL=0
MOVL C01544 V=800.0 PL=0
MOVL C01545 V=800.0 PL=0
MOVL C01546 V=800.0 PL=0
MOVL C01547 V=800.0 PL=0
MOVL C01548 V=800.0 PL=0
MOVL C01549 V=800.0 PL=0
MOVL C01550 V=800.0 PL=0
MOVL C01551 V=800.0 PL=0
MOVL C01552 V=800.0 PL=0
MOVL C01553 V=800.0 PL=0
MOVL C01554 V=800.0 PL=0
MOVL C01555 V=800.0 PL=0
MOVL C01556 V=800.0 PL=0
MOVL C01557 V=800.0 PL=0
MOVL C01558 V=800.0 PL=0
MOVL C01559 V=800.0 PL=0
MOVL C01560 V=800.0 PL=0
MOVL C01561 V=800.0 PL=0
MOVL C01562 V=800.0 PL=0
MOVL C01563 V=800.0 PL=0
MOVL C01564 V=800.0 PL=0
MOVL C01565 V=800.0 PL=0
MOVL C01566 V=800.0 PL=0
MOVL C01567 V=800.0 PL=0
MOVL C01568 V=800.0 PL=0
MOVL C01569 V=800.0 PL=0
MOVL C01570 V=800.0 PL=0
MOVL C01571 V=800.0 PL=0
MOVL C01572 V=800.0 PL=0
MOVL C01573 V=800.0 PL=0
MOVL C01574 V=800.0 PL=0
MOVL C01575 V=800.0 PL=0
MOVL C01576 V=800.0 PL=0
MOVL C01577 V=800.0 PL=0
MOVL C01578 V=800.0 PL=0
MOVL C01579 V=800.0 PL=0
MOVL C01580 V=800.0 PL=0
MOVL C01581 V=800.0 PL=0
MOVL C01582 V=800.0 PL=0
MOVL C01583 V=800.0 PL=0
MOVL C01584 V=800.0 PL=0
MOVL C01585 V=800.0 PL=0
MOVL C01586 V=800.0 PL=0
MOVL C01587 V=800.0 PL=0
MOVL C01588 V=800.0 PL=0
MOVL C01589 V=800.0 PL=0
MOVL C01590 V=800.0 PL=0
MOVL C01591 V=800.0 PL=0
MOVL C01592 V=800.0 PL=0
MOVL C01593 V=800.0 PL=0
MOVL C01594 V=800.0 PL=0
MOVL C01595 V=800.0 PL=0
MOVL C01596 V=800.0 PL=0
MOVL C01597 V=800.0 PL=0
MOVL C01598 V=800.0 PL=0
MOVL C01599 V=800.0 PL=0
MOVL C01600 V=800.0 PL=0
MOVL C01601 V=800.0 PL=0
MOVL C01602 V=800.0 PL=0
MOVL C01603 V=800.0 PL=0
MOVL C01604 V=800.0 PL=0
MOVL C01605 V=800.0 PL=0
MOVL C01606 V=800.0 PL=0
MOVL C01607 V=800.0 PL=0
MOVL C01608 V=800.0 PL=0
MOVL C01609 V=800.0 PL=0
MOVL C01610 V=800.0 PL=0
MOVL C01611 V=800.0 PL=0
MOVL C01612 V=800.0 PL=0
MOVL C01613 V=800.0 PL=0
MOVL C01614 V=800.0 PL=0
MOVL C01615 V=800.0 PL=0
MOVL C01616 V=800.0 PL=0
MOVL C01617 V=800.0 PL=0
MOVL C01618 V=800.0 PL=0
MOVL C01619 V=800.0 PL=0
MOVL C01620 V=800.0 PL=0
MOVL C01621 V=800.0 PL=0
MOVL C01622 V=800.0 PL=0
MOVL C01623 V=800.0 PL=0
MOVL C01624 V=800.0 PL=0
MOVL C01625 V=800.0 PL=0
MOVL C01626 V=800.0 PL=0
MOVL C01627 V=800.0 PL=0
MOVL C01628 V=800.0 PL=0
MOVL C01629 V=800.0 PL=0
MOVL C01630 V=800.0 PL=0
MOVL C01631 V=800.0 PL=0
MOVL C01632 V=800.0 PL=0
MOVL C01633 V=800.0 PL=0
MOVL C01634 V=800.0 PL=0
MOVL C01635 V=800.0 PL=0
MOVL C01636 V=800.0 PL=0
MOVL C01637 V=800.0 PL=0
MOVL C01638 V=800.0 PL=0
MOVL C01639 V=800.0 PL=0
MOVL C01640 V=800.0 PL=0
MOVL C01641 V=800.0 PL=0
MOVL C01642 V=800.0 PL=0
MOVL C01643 V=800.0 PL=0
MOVL C01644 V=800.0 PL=0
MOVL C01645 V=800.0 PL=0
MOVL C01646 V=800.0 PL=0
MOVL C01647 V=800.0 PL=0
MOVL C01648 V=800.0 PL=0
MOVL C01649 V=800.0 PL=0
MOVL C01650 V=800.0 PL=0
MOVL C01651 V=800.0 PL=0
MOVL C01652 V=800.0 PL=0
MOVL C01653 V=800.0 PL=0
MOVL C01654 V=800.0 PL=0
MOVL C01655 V=800.0 PL=0
MOVL C01656 V=800.0 PL=0
MOVL C01657 V=800.0 PL=0
MOVL C01658 V=800.0 PL=0
MOVL C01659 V=800.0 PL=0
MOVL C01660 V=800.0 PL=0
MOVL C01661 V=800.0 PL=0
MOVL C01662 V=800.0 PL=0
MOVL C01663 V=800.0 PL=0
MOVL C01664 V=800.0 PL=0
MOVL C01665 V=800.0 PL=0
MOVL C01666 V=800.0 PL=0
MOVL C01667 V=800.0 PL=0
MOVL C01668 V=800.0 PL=0
MOVL C01669 V=800.0 PL=0
MOVL C01670 V=800.0 PL=0
MOVL C01671 V=800.0 PL=0
MOVL C01672 V=800.0 PL=0
MOVL C01673 V=800.0 PL=0
MOVL C01674 V=800.0 PL=0
MOVL C01675 V=800.0 PL=0
MOVL C01676 V=800.0 PL=0
MOVL C01677 V=800.0 PL=0
MOVL C01678 V=800.0 PL=0
MOVL C01679 V=800.0 PL=0
MOVL C01680 V=800.0 PL=0
MOVL C01681 V=800.0 PL=0
MOVL C01682 V=800.0 PL=0
MOVL C01683 V=800.0 PL=0
MOVL C01684 V=800.0 PL=0
MOVL C01685 V=800.0 PL=0
MOVL C01686 V=800.0 PL=0
MOVL C01687 V=800.0 PL=0
MOVL C01688 V=800.0 PL=0
MOVL C01689 V=800.0 PL=0
MOVL C01690 V=800.0 PL=0
MOVL C01691 V=800.0 PL=0
MOVL C01692 V=800.0 PL=0
MOVL C01693 V=800.0 PL=0
MOVL C01694 V=800.0 PL=0
MOVL C01695 V=800.0 PL=0
MOVL C01696 V=800.0 PL=0
MOVL C01697 V=800.0 PL=0
MOVL C01698 V=800.0 PL=0
MOVL C01699 V=800.0 PL=0
MOVL C01700 V=800.0 PL=0
MOVL C01701 V=800.0 PL=0
MOVL C01702 V=800.0 PL=0
MOVL C01703 V=800.0 PL=0
MOVL C01704 V=800.0 PL=0
MOVL C01705 V=800.0 PL=0
MOVL C01706 V=800.0 PL=0
MOVL C01707 V=800.0 PL=0
MOVL C01708 V=800.0 PL=0
MOVL C01709 V=800.0 PL=0
MOVL C01710 V=800.0 PL=0
MOVL C01711 V=800.0 PL=0
MOVL C01712 V=800.0 PL=0
MOVL C01713 V=800.0 PL=0
MOVL C01714 V=800.0 PL=0
MOVL C01715 V=800.0 PL=0
MOVL C01716 V=800.0 PL=0
MOVL C01717 V=800.0 PL=0
MOVL C01718 V=800.0 PL=0
MOVL C01719 V=800.0 PL=0
MOVL C01720 V=800.0 PL=0
MOVL C01721 V=800.0 PL=0
MOVL C01722 V=800.0 PL=0
MOVL C01723 V=800.0 PL=0
MOVL C01724 V=800.0 PL=0
MOVL C01725 V=800.0 PL=0
MOVL C01726 V=800.0 PL=0
MOVL C01727 V=800.0 PL=0
MOVL C01728 V=800.0 PL=0
MOVL C01729 V=800.0 PL=0
MOVL C01730 V=800.0 PL=0
MOVL C01731 V=800.0 PL=0
MOVL C01732 V=800.0 PL=0
MOVL C01733 V=800.0 PL=0
MOVL C01734 V=800.0 PL=0
MOVL C01735 V=800.0 PL=0
MOVL C01736 V=800.0 PL=0
MOVL C01737 V=800.0 PL=0
MOVL C01738 V=800.0 PL=0
MOVL C01739 V=800.0 PL=0
MOVL C01740 V=800.0 PL=0
MOVL C01741 V=800.0 PL=0
MOVL C01742 V=800.0 PL=0
MOVL C01743 V=800.0 PL=0
MOVL C01744 V=800.0 PL=0
MOVL C01745 V=800.0 PL=0
MOVL C01746 V=800.0 PL=0
MOVL C01747 V=800.0 PL=0
MOVL C01748 V=800.0 PL=0
MOVL C01749 V=800.0 PL=0
MOVL C01750 V=800.0 PL=0
MOVL C01751 V=800.0 PL=0
MOVL C01752 V=800.0 PL=0
MOVL C01753 V=800.0 PL=0
MOVL C01754 V=800.0 PL=0
MOVL C01755 V=800.0 PL=0
MOVL C01756 V=800.0 PL=0
MOVL C01757 V=800.0 PL=0
MOVL C01758 V=800.0 PL=0
MOVL C01759 V=800.0 PL=0
MOVL C01760 V=800.0 PL=0
MOVL C01761 V=800.0 PL=0
MOVL C01762 V=800.0 PL=0
MOVL C01763 V=800.0 PL=0
MOVL C01764 V=800.0 PL=0
MOVL C01765 V=800.0 PL=0
MOVL C01766 V=800.0 PL=0
MOVL C01767 V=800.0 PL=0
MOVL C01768 V=800.0 PL=0
MOVL C01769 V=800.0 PL=0
MOVL C01770 V=800.0 PL=0
MOVL C01771 V=800.0 PL=0
MOVL C01772 V=800.0 PL=0
MOVL C01773 V=800.0 PL=0
MOVL C01774 V=800.0 PL=0
MOVL C01775 V=800.0 PL=0
MOVL C01776 V=800.0 PL=0
MOVL C01777 V=800.0 PL=0
MOVL C01778 V=800.0 PL=0
MOVL C01779 V=800.0 PL=0
MOVL C01780 V=800.0 PL=0
MOVL C01781 V=800.0 PL=0
MOVL C01782 V=800.0 PL=0
MOVL C01783 V=800.0 PL=0
MOVL C01784 V=800.0 PL=0
MOVL C01785 V=800.0 PL=0
MOVL C01786 V=800.0 PL=0
MOVL C01787 V=800.0 PL=0
MOVL C01788 V=800.0 PL=0
MOVL C01789 V=800.0 PL=0
MOVL C01790 V=800.0 PL=0
MOVL C01791 V=800.0 PL=0
MOVL C01792 V=800.0 PL=0
MOVL C01793 V=800.0 PL=0
MOVL C01794 V=800.0 PL=0
MOVL C01795 V=800.0 PL=0
MOVL C01796 V=800.0 PL=0
MOVL C01797 V=800.0 PL=0
MOVL C01798 V=800.0 PL=0
MOVL C01799 V=800.0 PL=0
MOVL C01800 V=800.0 PL=0
MOVL C01801 V=800.0 PL=0
MOVL C01802 V=800.0 PL=0
MOVL C01803 V=800.0 PL=0
MOVL C01804 V=800.0 PL=0
MOVL C01805 V=800.0 PL=0
MOVL C01806 V=800.0 PL=0
MOVL C01807 V=800.0 PL=0
MOVL C01808 V=800.0 PL=0
MOVL C01809 V=800.0 PL=0
MOVL C01810 V=800.0 PL=0
MOVL C01811 V=800.0 PL=0
MOVL C01812 V=800.0 PL=0
MOVL C01813 V=800.0 PL=0
MOVL C01814 V=800.0 PL=0
MOVL C01815 V=800.0 PL=0
MOVL C01816 V=800.0 PL=0
MOVL C01817 V=800.0 PL=0
MOVL C01818 V=800.0 PL=0
MOVL C01819 V=800.0 PL=0
MOVL C01820 V=800.0 PL=0
MOVL C01821 V=800.0 PL=0
MOVL C01822 V=800.0 PL=0
MOVL C01823 V=800.0 PL=0
MOVL C01824 V=800.0 PL=0
MOVL C01825 V=800.0 PL=0
MOVL C01826 V=800.0 PL=0
MOVL C01827 V=800.0 PL=0
MOVL C01828 V=800.0 PL=0
MOVL C01829 V=800.0 PL=0
MOVL C01830 V=800.0 PL=0
MOVL C01831 V=800.0 PL=0
MOVL C01832 V=800.0 PL=0
MOVL C01833 V=800.0 PL=0
MOVL C01834 V=800.0 PL=0
MOVL C01835 V=800.0 PL=0
MOVL C01836 V=800.0 PL=0
MOVL C01837 V=800.0 PL=0
MOVL C01838 V=800.0 PL=0
MOVL C01839 V=800.0 PL=0
MOVL C01840 V=800.0 PL=0
MOVL C01841 V=800.0 PL=0
MOVL C01842 V=800.0 PL=0
MOVL C01843 V=800.0 PL=0
MOVL C01844 V=800.0 PL=0
MOVL C01845 V=800.0 PL=0
MOVL C01846 V=800.0 PL=0
MOVL C01847 V=800.0 PL=0
MOVL C01848 V=800.0 PL=0
MOVL C01849 V=800.0 PL=0
MOVL C01850 V=800.0 PL=0
MOVL C01851 V=800.0 PL=0
MOVL C01852 V=800.0 PL=0
MOVL C01853 V=800.0 PL=0
MOVL C01854 V=800.0 PL=0
MOVL C01855 V=800.0 PL=0
MOVL C01856 V=800.0 PL=0
MOVL C01857 V=800.0 PL=0
MOVL C01858 V=800.0 PL=0
MOVL C01859 V=800.0 PL=0
MOVL C01860 V=800.0 PL=0
MOVL C01861 V=800.0 PL=0
MOVL C01862 V=800.0 PL=0
MOVL C01863 V=800.0 PL=0
MOVL C01864 V=800.0 PL=0
MOVL C01865 V=800.0 PL=0
MOVL C01866 V=800.0 PL=0
MOVL C01867 V=800.0 PL=0
MOVL C01868 V=800.0 PL=0
MOVL C01869 V=800.0 PL=0
MOVL C01870 V=800.0 PL=0
MOVL C01871 V=800.0 PL=0
MOVL C01872 V=800.0 PL=0
MOVL C01873 V=800.0 PL=0
MOVL C01874 V=800.0 PL=0
MOVL C01875 V=800.0 PL=0
MOVL C01876 V=800.0 PL=0
MOVL C01877 V=800.0 PL=0
MOVL C01878 V=800.0 PL=0
MOVL C01879 V=800.0 PL=0
MOVL C01880 V=800.0 PL=0
MOVL C01881 V=800.0 PL=0
MOVL C01882 V=800.0 PL=0
MOVL C01883 V=800.0 PL=0
MOVL C01884 V=800.0 PL=0
MOVL C01885 V=800.0 PL=0
MOVL C01886 V=800.0 PL=0
MOVL C01887 V=800.0 PL=0
MOVL C01888 V=800.0 PL=0
MOVL C01889 V=800.0 PL=0
MOVL C01890 V=800.0 PL=0
MOVL C01891 V=800.0 PL=0
MOVL C01892 V=800.0 PL=0
MOVL C01893 V=800.0 PL=0
MOVL C01894 V=800.0 PL=0
MOVL C01895 V=800.0 PL=0
MOVL C01896 V=800.0 PL=0
MOVL C01897 V=800.0 PL=0
MOVL C01898 V=800.0 PL=0
MOVL C01899 V=800.0 PL=0
MOVL C01900 V=800.0 PL=0
MOVL C01901 V=800.0 PL=0
MOVL C01902 V=800.0 PL=0
MOVL C01903 V=800.0 PL=0
MOVL C01904 V=800.0 PL=0
MOVL C01905 V=800.0 PL=0
MOVL C01906 V=800.0 PL=0
MOVL C01907 V=800.0 PL=0
MOVL C01908 V=800.0 PL=0
MOVL C01909 V=800.0 PL=0
MOVL C01910 V=800.0 PL=0
MOVL C01911 V=800.0 PL=0
MOVL C01912 V=800.0 PL=0
MOVL C01913 V=800.0 PL=0
MOVL C01914 V=800.0 PL=0
MOVL C01915 V=800.0 PL=0
MOVL C01916 V=800.0 PL=0
MOVL C01917 V=800.0 PL=0
MOVL C01918 V=800.0 PL=0
MOVL C01919 V=800.0 PL=0
MOVL C01920 V=800.0 PL=0
MOVL C01921 V=800.0 PL=0
MOVL C01922 V=800.0 PL=0
MOVL C01923 V=800.0 PL=0
MOVL C01924 V=800.0 PL=0
MOVL C01925 V=800.0 PL=0
MOVL C01926 V=800.0 PL=0
MOVL C01927 V=800.0 PL=0
MOVL C01928 V=800.0 PL=0
MOVL C01929 V=800.0 PL=0
MOVL C01930 V=800.0 PL=0
MOVL C01931 V=800.0 PL=0
MOVL C01932 V=800.0 PL=0
MOVL C01933 V=800.0 PL=0
MOVL C01934 V=800.0 PL=0
MOVL C01935 V=800.0 PL=0
MOVL C01936 V=800.0 PL=0
MOVL C01937 V=800.0 PL=0
MOVL C01938 V=800.0 PL=0
MOVL C01939 V=800.0 PL=0
MOVL C01940 V=800.0 PL=0
MOVL C01941 V=800.0 PL=0
MOVL C01942 V=800.0 PL=0
MOVL C01943 V=800.0 PL=0
MOVL C01944 V=800.0 PL=0
MOVL C01945 V=800.0 PL=0
MOVL C01946 V=800.0 PL=0
MOVL C01947 V=800.0 PL=0
MOVL C01948 V=800.0 PL=0
MOVL C01949 V=800.0 PL=0
MOVL C01950 V=800.0 PL=0
MOVL C01951 V=800.0 PL=0
MOVL C01952 V=800.0 PL=0
MOVL C01953 V=800.0 PL=0
MOVL C01954 V=800.0 PL=0
MOVL C01955 V=800.0 PL=0
MOVL C01956 V=800.0 PL=0
MOVL C01957 V=800.0 PL=0
MOVL C01958 V=800.0 PL=0
MOVL C01959 V=800.0 PL=0
MOVL C01960 V=800.0 PL=0
MOVL C01961 V=800.0 PL=0
MOVL C01962 V=800.0 PL=0
MOVL C01963 V=800.0 PL=0
MOVL C01964 V=800.0 PL=0
MOVL C01965 V=800.0 PL=0
MOVL C01966 V=800.0 PL=0
MOVL C01967 V=800.0 PL=0
MOVL C01968 V=800.0 PL=0
MOVL C01969 V=800.0 PL=0
MOVL C01970 V=800.0 PL=0
MOVL C01971 V=800.0 PL=0
MOVL C01972 V=800.0 PL=0
MOVL C01973 V=800.0 PL=0
MOVL C01974 V=800.0 PL=0
MOVL C01975 V=800.0 PL=0
MOVL C01976 V=800.0 PL=0
MOVL C01977 V=800.0 PL=0
MOVL C01978 V=800.0 PL=0
MOVL C01979 V=800.0 PL=0
MOVL C01980 V=800.0 PL=0
MOVL C01981 V=800.0 PL=0
MOVL C01982 V=800.0 PL=0
MOVL C01983 V=800.0 PL=0
MOVL C01984 V=800.0 PL=0
MOVL C01985 V=800.0 PL=0
MOVL C01986 V=800.0 PL=0
MOVL C01987 V=800.0 PL=0
MOVL C01988 V=800.0 PL=0
MOVL C01989 V=800.0 PL=0
MOVL C01990 V=800.0 PL=0
MOVL C01991 V=800.0 PL=0
MOVL C01992 V=800.0 PL=0
MOVL C01993 V=800.0 PL=0
MOVL C01994 V=800.0 PL=0
MOVL C01995 V=800.0 PL=0
MOVL C01996 V=800.0 PL=0
MOVL C01997 V=800.0 PL=0
MOVL C01998 V=800.0 PL=0
MOVL C01999 V=800.0 PL=0
MOVL C02000 V=800.0 PL=0
MOVL C02001 V=800.0 PL=0
MOVL C02002 V=800.0 PL=0
MOVL C02003 V=800.0 PL=0
MOVL C02004 V=800.0 PL=0
MOVL C02005 V=800.0 PL=0
MOVL C02006 V=800.0 PL=0
MOVL C02007 V=800.0 PL=0
MOVL C02008 V=800.0 PL=0
MOVL C02009 V=800.0 PL=0
MOVL C02010 V=800.0 PL=0
MOVL C02011 V=800.0 PL=0
MOVL C02012 V=800.0 PL=0
MOVL C02013 V=800.0 PL=0
MOVL C02014 V=800.0 PL=0
MOVL C02015 V=800.0 PL=0
MOVL C02016 V=800.0 PL=0
MOVL C02017 V=800.0 PL=0
MOVL C02018 V=800.0 PL=0
MOVL C02019 V=800.0 PL=0
MOVL C02020 V=800.0 PL=0
MOVL C02021 V=800.0 PL=0
MOVL C02022 V=800.0 PL=0
MOVL C02023 V=800.0 PL=0
MOVL C02024 V=800.0 PL=0
MOVL C02025 V=800.0 PL=0
MOVL C02026 V=800.0 PL=0
MOVL C02027 V=800.0 PL=0
MOVL C02028 V=800.0 PL=0
MOVL C02029 V=800.0 PL=0
MOVL C02030 V=800.0 PL=0
MOVL C02031 V=800.0 PL=0
MOVL C02032 V=800.0 PL=0
MOVL C02033 V=800.0 PL=0
MOVL C02034 V=800.0 PL=0
MOVL C02035 V=800.0 PL=0
MOVL C02036 V=800.0 PL=0
MOVL C02037 V=800.0 PL=0
MOVL C02038 V=800.0 PL=0
MOVL C02039 V=800.0 PL=0
MOVL C02040 V=800.0 PL=0
MOVL C02041 V=800.0 PL=0
MOVL C02042 V=800.0 PL=0
MOVL C02043 V=800.0 PL=0
MOVL C02044 V=800.0 PL=0
MOVL C02045 V=800.0 PL=0
MOVL C02046 V=800.0 PL=0
MOVL C02047 V=800.0 PL=0
MOVL C02048 V=800.0 PL=0
MOVL C02049 V=800.0 PL=0
MOVL C02050 V=800.0 PL=0
MOVL C02051 V=800.0 PL=0
MOVL C02052 V=800.0 PL=0
MOVL C02053 V=800.0 PL=0
MOVL C02054 V=800.0 PL=0
MOVL C02055 V=800.0 PL=0
MOVL C02056 V=800.0 PL=0
MOVL C02057 V=800.0 PL=0
MOVL C02058 V=800.0 PL=0
MOVL C02059 V=800.0 PL=0
MOVL C02060 V=800.0 PL=0
MOVL C02061 V=800.0 PL=0
MOVL C02062 V=800.0 PL=0
MOVL C02063 V=800.0 PL=0
MOVL C02064 V=800.0 PL=0
MOVL C02065 V=800.0 PL=0
MOVL C02066 V=800.0 PL=0
MOVL C02067 V=800.0 PL=0
MOVL C02068 V=800.0 PL=0
MOVL C02069 V=800.0 PL=0
MOVL C02070 V=800.0 PL=0
MOVL C02071 V=800.0 PL=0
MOVL C02072 V=800.0 PL=0
MOVL C02073 V=800.0 PL=0
MOVL C02074 V=800.0 PL=0
MOVL C02075 V=800.0 PL=0
MOVL C02076 V=800.0 PL=0
MOVL C02077 V=800.0 PL=0
MOVL C02078 V=800.0 PL=0
MOVL C02079 V=800.0 PL=0
MOVL C02080 V=800.0 PL=0
MOVL C02081 V=800.0 PL=0
MOVL C02082 V=800.0 PL=0
MOVL C02083 V=800.0 PL=0
MOVL C02084 V=800.0 PL=0
MOVL C02085 V=800.0 PL=0
MOVL C02086 V=800.0 PL=0
MOVL C02087 V=800.0 PL=0
MOVL C02088 V=800.0 PL=0
MOVL C02089 V=800.0 PL=0
MOVL C02090 V=800.0 PL=0
MOVL C02091 V=800.0 PL=0
MOVL C02092 V=800.0 PL=0
MOVL C02093 V=800.0 PL=0
MOVL C02094 V=800.0 PL=0
MOVL C02095 V=800.0 PL=0
MOVL C02096 V=800.0 PL=0
MOVL C02097 V=800.0 PL=0
MOVL C02098 V=800.0 PL=0
MOVL C02099 V=800.0 PL=0
MOVL C02100 V=800.0 PL=0
MOVL C02101 V=800.0 PL=0
MOVL C02102 V=800.0 PL=0
MOVL C02103 V=800.0 PL=0
MOVL C02104 V=800.0 PL=0
MOVL C02105 V=800.0 PL=0
MOVL C02106 V=800.0 PL=0
MOVL C02107 V=800.0 PL=0
MOVL C02108 V=800.0 PL=0
MOVL C02109 V=800.0 PL=0
MOVL C02110 V=800.0 PL=0
MOVL C02111 V=800.0 PL=0
MOVL C02112 V=800.0 PL=0
MOVL C02113 V=800.0 PL=0
MOVL C02114 V=800.0 PL=0
MOVL C02115 V=800.0 PL=0
MOVL C02116 V=800.0 PL=0
